    TriggL T0,v50,laserON,z0,toolEtna\WObj:=wobjEtna;
    TriggL T1,vl,laserOFF,z0,toolEtna\WObj:=wobjEtna;
    TriggL T2,v50,laserON,z0,toolEtna\WObj:=wobjEtna;
    TriggL T3,vl,laserOFF,z0,toolEtna\WObj:=wobjEtna;
    TriggL T4,v50,laserON,z0,toolEtna\WObj:=wobjEtna;
    TriggL T5,vl,laserOFF,z0,toolEtna\WObj:=wobjEtna;
    TriggL T6,v50,laserON,z0,toolEtna\WObj:=wobjEtna;
    TriggL T7,vl,laserOFF,z0,toolEtna\WObj:=wobjEtna;
    TriggL T8,v50,laserON,z0,toolEtna\WObj:=wobjEtna;
    TriggL T9,vl,laserOFF,z0,toolEtna\WObj:=wobjEtna;
    TriggL T10,v50,laserON,z0,toolEtna\WObj:=wobjEtna;
    TriggL T11,vl,laserOFF,z0,toolEtna\WObj:=wobjEtna;
    TriggL T12,v50,laserON,z0,toolEtna\WObj:=wobjEtna;
    TriggL T13,vl,laserOFF,z0,toolEtna\WObj:=wobjEtna;
    TriggL T14,v50,laserON,z0,toolEtna\WObj:=wobjEtna;
    TriggL T15,vl,laserOFF,z0,toolEtna\WObj:=wobjEtna;
    TriggL T16,v50,laserON,z0,toolEtna\WObj:=wobjEtna;
    TriggL T17,vl,laserOFF,z0,toolEtna\WObj:=wobjEtna;
    TriggL T18,v50,laserON,z0,toolEtna\WObj:=wobjEtna;
    TriggL T19,vl,laserOFF,z0,toolEtna\WObj:=wobjEtna;
    TriggL T20,v50,laserON,z0,toolEtna\WObj:=wobjEtna;
    TriggL T21,vl,laserOFF,z0,toolEtna\WObj:=wobjEtna;
    TriggL T22,v50,laserON,z0,toolEtna\WObj:=wobjEtna;
    TriggL T23,vl,laserOFF,z0,toolEtna\WObj:=wobjEtna;
    TriggL T24,v50,laserON,z0,toolEtna\WObj:=wobjEtna;
    TriggL T25,vl,laserOFF,z0,toolEtna\WObj:=wobjEtna;
    TriggL T26,v50,laserON,z0,toolEtna\WObj:=wobjEtna;
    TriggL T27,vl,laserOFF,z0,toolEtna\WObj:=wobjEtna;
    TriggL T28,v50,laserON,z0,toolEtna\WObj:=wobjEtna;
    TriggL T29,vl,laserOFF,z0,toolEtna\WObj:=wobjEtna;
    TriggL T30,v50,laserON,z0,toolEtna\WObj:=wobjEtna;
    TriggL T31,vl,laserOFF,z0,toolEtna\WObj:=wobjEtna;
    TriggL T32,v50,laserON,z0,toolEtna\WObj:=wobjEtna;
    TriggL T33,vl,laserOFF,z0,toolEtna\WObj:=wobjEtna;
    TriggL T34,v50,laserON,z0,toolEtna\WObj:=wobjEtna;
    TriggL T35,vl,laserOFF,z0,toolEtna\WObj:=wobjEtna;
    TriggL T36,v50,laserON,z0,toolEtna\WObj:=wobjEtna;
    TriggL T37,vl,laserOFF,z0,toolEtna\WObj:=wobjEtna;
    TriggL T38,v50,laserON,z0,toolEtna\WObj:=wobjEtna;
    TriggL T39,vl,laserOFF,z0,toolEtna\WObj:=wobjEtna;
    TriggL T40,v50,laserON,z0,toolEtna\WObj:=wobjEtna;
    TriggL T41,vl,laserOFF,z0,toolEtna\WObj:=wobjEtna;
    TriggL T42,v50,laserON,z0,toolEtna\WObj:=wobjEtna;
    TriggL T43,vl,laserOFF,z0,toolEtna\WObj:=wobjEtna;
    TriggL T44,v50,laserON,z0,toolEtna\WObj:=wobjEtna;
    TriggL T45,vl,laserOFF,z0,toolEtna\WObj:=wobjEtna;
    TriggL T46,v50,laserON,z0,toolEtna\WObj:=wobjEtna;
    TriggL T47,vl,laserOFF,z0,toolEtna\WObj:=wobjEtna;
    TriggL T48,v50,laserON,z0,toolEtna\WObj:=wobjEtna;
    TriggL T49,vl,laserOFF,z0,toolEtna\WObj:=wobjEtna;
    TriggL T50,v50,laserON,z0,toolEtna\WObj:=wobjEtna;
    TriggL T51,vl,laserOFF,z0,toolEtna\WObj:=wobjEtna;
    TriggL T52,v50,laserON,z0,toolEtna\WObj:=wobjEtna;
    TriggL T53,vl,laserOFF,z0,toolEtna\WObj:=wobjEtna;
    TriggL T54,v50,laserON,z0,toolEtna\WObj:=wobjEtna;
    TriggL T55,vl,laserOFF,z0,toolEtna\WObj:=wobjEtna;
    TriggL T56,v50,laserON,z0,toolEtna\WObj:=wobjEtna;
    TriggL T57,vl,laserOFF,z0,toolEtna\WObj:=wobjEtna;
    TriggL T58,v50,laserON,z0,toolEtna\WObj:=wobjEtna;
    TriggL T59,vl,laserOFF,z0,toolEtna\WObj:=wobjEtna;
    TriggL T60,v50,laserON,z0,toolEtna\WObj:=wobjEtna;
    TriggL T61,vl,laserOFF,z0,toolEtna\WObj:=wobjEtna;
    TriggL T62,v50,laserON,z0,toolEtna\WObj:=wobjEtna;
    TriggL T63,vl,laserOFF,z0,toolEtna\WObj:=wobjEtna;
    TriggL T64,v50,laserON,z0,toolEtna\WObj:=wobjEtna;
    TriggL T65,vl,laserOFF,z0,toolEtna\WObj:=wobjEtna;
    TriggL T66,v50,laserON,z0,toolEtna\WObj:=wobjEtna;
    TriggL T67,vl,laserOFF,z0,toolEtna\WObj:=wobjEtna;
    TriggL T68,v50,laserON,z0,toolEtna\WObj:=wobjEtna;
    TriggL T69,vl,laserOFF,z0,toolEtna\WObj:=wobjEtna;
    TriggL T70,v50,laserON,z0,toolEtna\WObj:=wobjEtna;
    TriggL T71,vl,laserOFF,z0,toolEtna\WObj:=wobjEtna;
    TriggL T72,v50,laserON,z0,toolEtna\WObj:=wobjEtna;
    TriggL T73,vl,laserOFF,z0,toolEtna\WObj:=wobjEtna;
    TriggL T74,v50,laserON,z0,toolEtna\WObj:=wobjEtna;
    TriggL T75,vl,laserOFF,z0,toolEtna\WObj:=wobjEtna;
    TriggL T76,v50,laserON,z0,toolEtna\WObj:=wobjEtna;
    TriggL T77,vl,laserOFF,z0,toolEtna\WObj:=wobjEtna;
    TriggL T78,v50,laserON,z0,toolEtna\WObj:=wobjEtna;
    TriggL T79,vl,laserOFF,z0,toolEtna\WObj:=wobjEtna;
    TriggL T80,v50,laserON,z0,toolEtna\WObj:=wobjEtna;
    TriggL T81,vl,laserOFF,z0,toolEtna\WObj:=wobjEtna;
    TriggL T82,v50,laserON,z0,toolEtna\WObj:=wobjEtna;
    TriggL T83,vl,laserOFF,z0,toolEtna\WObj:=wobjEtna;
    TriggL T84,v50,laserON,z0,toolEtna\WObj:=wobjEtna;
    TriggL T85,vl,laserOFF,z0,toolEtna\WObj:=wobjEtna;
    TriggL T86,v50,laserON,z0,toolEtna\WObj:=wobjEtna;
    TriggL T87,vl,laserOFF,z0,toolEtna\WObj:=wobjEtna;
    TriggL T88,v50,laserON,z0,toolEtna\WObj:=wobjEtna;
    TriggL T89,vl,laserOFF,z0,toolEtna\WObj:=wobjEtna;
    TriggL T90,v50,laserON,z0,toolEtna\WObj:=wobjEtna;
    TriggL T91,vl,laserOFF,z0,toolEtna\WObj:=wobjEtna;
    TriggL T92,v50,laserON,z0,toolEtna\WObj:=wobjEtna;
    TriggL T93,vl,laserOFF,z0,toolEtna\WObj:=wobjEtna;
    TriggL T94,v50,laserON,z0,toolEtna\WObj:=wobjEtna;
    TriggL T95,vl,laserOFF,z0,toolEtna\WObj:=wobjEtna;
    TriggL T96,v50,laserON,z0,toolEtna\WObj:=wobjEtna;
    TriggL T97,vl,laserOFF,z0,toolEtna\WObj:=wobjEtna;
    TriggL T98,v50,laserON,z0,toolEtna\WObj:=wobjEtna;
    TriggL T99,vl,laserOFF,z0,toolEtna\WObj:=wobjEtna;
    TriggL T100,v50,laserON,z0,toolEtna\WObj:=wobjEtna;
    TriggL T101,vl,laserOFF,z0,toolEtna\WObj:=wobjEtna;
    TriggL T102,v50,laserON,z0,toolEtna\WObj:=wobjEtna;
    TriggL T103,vl,laserOFF,z0,toolEtna\WObj:=wobjEtna;
    TriggL T104,v50,laserON,z0,toolEtna\WObj:=wobjEtna;
    TriggL T105,vl,laserOFF,z0,toolEtna\WObj:=wobjEtna;
    TriggL T106,v50,laserON,z0,toolEtna\WObj:=wobjEtna;
    TriggL T107,vl,laserOFF,z0,toolEtna\WObj:=wobjEtna;
    TriggL T108,v50,laserON,z0,toolEtna\WObj:=wobjEtna;
    TriggL T109,vl,laserOFF,z0,toolEtna\WObj:=wobjEtna;
    TriggL T110,v50,laserON,z0,toolEtna\WObj:=wobjEtna;
    TriggL T111,vl,laserOFF,z0,toolEtna\WObj:=wobjEtna;
    TriggL T112,v50,laserON,z0,toolEtna\WObj:=wobjEtna;
    TriggL T113,vl,laserOFF,z0,toolEtna\WObj:=wobjEtna;
    TriggL T114,v50,laserON,z0,toolEtna\WObj:=wobjEtna;
    TriggL T115,vl,laserOFF,z0,toolEtna\WObj:=wobjEtna;
    TriggL T116,v50,laserON,z0,toolEtna\WObj:=wobjEtna;
    TriggL T117,vl,laserOFF,z0,toolEtna\WObj:=wobjEtna;
    TriggL T118,v50,laserON,z0,toolEtna\WObj:=wobjEtna;
    TriggL T119,vl,laserOFF,z0,toolEtna\WObj:=wobjEtna;
    TriggL T120,v50,laserON,z0,toolEtna\WObj:=wobjEtna;
    TriggL T121,vl,laserOFF,z0,toolEtna\WObj:=wobjEtna;
    TriggL T122,v50,laserON,z0,toolEtna\WObj:=wobjEtna;
    TriggL T123,vl,laserOFF,z0,toolEtna\WObj:=wobjEtna;
    TriggL T124,v50,laserON,z0,toolEtna\WObj:=wobjEtna;
    TriggL T125,vl,laserOFF,z0,toolEtna\WObj:=wobjEtna;
    TriggL T126,v50,laserON,z0,toolEtna\WObj:=wobjEtna;
    TriggL T127,vl,laserOFF,z0,toolEtna\WObj:=wobjEtna;
    TriggL T128,v50,laserON,z0,toolEtna\WObj:=wobjEtna;
    TriggL T129,vl,laserOFF,z0,toolEtna\WObj:=wobjEtna;
    TriggL T130,v50,laserON,z0,toolEtna\WObj:=wobjEtna;
    TriggL T131,vl,laserOFF,z0,toolEtna\WObj:=wobjEtna;
    TriggL T132,v50,laserON,z0,toolEtna\WObj:=wobjEtna;
    TriggL T133,vl,laserOFF,z0,toolEtna\WObj:=wobjEtna;
    TriggL T134,v50,laserON,z0,toolEtna\WObj:=wobjEtna;
    TriggL T135,vl,laserOFF,z0,toolEtna\WObj:=wobjEtna;
    TriggL T136,v50,laserON,z0,toolEtna\WObj:=wobjEtna;
    TriggL T137,vl,laserOFF,z0,toolEtna\WObj:=wobjEtna;
    TriggL T138,v50,laserON,z0,toolEtna\WObj:=wobjEtna;
    TriggL T139,vl,laserOFF,z0,toolEtna\WObj:=wobjEtna;
    TriggL T140,v50,laserON,z0,toolEtna\WObj:=wobjEtna;
    TriggL T141,vl,laserOFF,z0,toolEtna\WObj:=wobjEtna;
    TriggL T142,v50,laserON,z0,toolEtna\WObj:=wobjEtna;
    TriggL T143,vl,laserOFF,z0,toolEtna\WObj:=wobjEtna;
    TriggL T144,v50,laserON,z0,toolEtna\WObj:=wobjEtna;
    TriggL T145,vl,laserOFF,z0,toolEtna\WObj:=wobjEtna;
    TriggL T146,v50,laserON,z0,toolEtna\WObj:=wobjEtna;
    TriggL T147,vl,laserOFF,z0,toolEtna\WObj:=wobjEtna;
    TriggL T148,v50,laserON,z0,toolEtna\WObj:=wobjEtna;
    TriggL T149,vl,laserOFF,z0,toolEtna\WObj:=wobjEtna;
    TriggL T150,v50,laserON,z0,toolEtna\WObj:=wobjEtna;
    TriggL T151,vl,laserOFF,z0,toolEtna\WObj:=wobjEtna;
    TriggL T152,v50,laserON,z0,toolEtna\WObj:=wobjEtna;
    TriggL T153,vl,laserOFF,z0,toolEtna\WObj:=wobjEtna;
    TriggL T154,v50,laserON,z0,toolEtna\WObj:=wobjEtna;
    TriggL T155,vl,laserOFF,z0,toolEtna\WObj:=wobjEtna;
    TriggL T156,v50,laserON,z0,toolEtna\WObj:=wobjEtna;
    TriggL T157,vl,laserOFF,z0,toolEtna\WObj:=wobjEtna;
    TriggL T158,v50,laserON,z0,toolEtna\WObj:=wobjEtna;
    TriggL T159,vl,laserOFF,z0,toolEtna\WObj:=wobjEtna;
    TriggL T160,v50,laserON,z0,toolEtna\WObj:=wobjEtna;
    TriggL T161,vl,laserOFF,z0,toolEtna\WObj:=wobjEtna;
    TriggL T162,v50,laserON,z0,toolEtna\WObj:=wobjEtna;
    TriggL T163,vl,laserOFF,z0,toolEtna\WObj:=wobjEtna;
    TriggL T164,v50,laserON,z0,toolEtna\WObj:=wobjEtna;
    TriggL T165,vl,laserOFF,z0,toolEtna\WObj:=wobjEtna;
    TriggL T166,v50,laserON,z0,toolEtna\WObj:=wobjEtna;
    TriggL T167,vl,laserOFF,z0,toolEtna\WObj:=wobjEtna;
    TriggL T168,v50,laserON,z0,toolEtna\WObj:=wobjEtna;
    TriggL T169,vl,laserOFF,z0,toolEtna\WObj:=wobjEtna;
    TriggL T170,v50,laserON,z0,toolEtna\WObj:=wobjEtna;
    TriggL T171,vl,laserOFF,z0,toolEtna\WObj:=wobjEtna;
    TriggL T172,v50,laserON,z0,toolEtna\WObj:=wobjEtna;
    TriggL T173,vl,laserOFF,z0,toolEtna\WObj:=wobjEtna;
    TriggL T174,v50,laserON,z0,toolEtna\WObj:=wobjEtna;
    TriggL T175,vl,laserOFF,z0,toolEtna\WObj:=wobjEtna;
    TriggL T176,v50,laserON,z0,toolEtna\WObj:=wobjEtna;
    TriggL T177,vl,laserOFF,z0,toolEtna\WObj:=wobjEtna;
    TriggL T178,v50,laserON,z0,toolEtna\WObj:=wobjEtna;
    TriggL T179,vl,laserOFF,z0,toolEtna\WObj:=wobjEtna;
    TriggL T180,v50,laserON,z0,toolEtna\WObj:=wobjEtna;
    TriggL T181,vl,laserOFF,z0,toolEtna\WObj:=wobjEtna;
    TriggL T182,v50,laserON,z0,toolEtna\WObj:=wobjEtna;
    TriggL T183,vl,laserOFF,z0,toolEtna\WObj:=wobjEtna;
    TriggL T184,v50,laserON,z0,toolEtna\WObj:=wobjEtna;
    TriggL T185,vl,laserOFF,z0,toolEtna\WObj:=wobjEtna;
    TriggL T186,v50,laserON,z0,toolEtna\WObj:=wobjEtna;
    TriggL T187,vl,laserOFF,z0,toolEtna\WObj:=wobjEtna;
    TriggL T188,v50,laserON,z0,toolEtna\WObj:=wobjEtna;
    TriggL T189,vl,laserOFF,z0,toolEtna\WObj:=wobjEtna;
    TriggL T190,v50,laserON,z0,toolEtna\WObj:=wobjEtna;
    TriggL T191,vl,laserOFF,z0,toolEtna\WObj:=wobjEtna;
    TriggL T192,v50,laserON,z0,toolEtna\WObj:=wobjEtna;
    TriggL T193,vl,laserOFF,z0,toolEtna\WObj:=wobjEtna;
    TriggL T194,v50,laserON,z0,toolEtna\WObj:=wobjEtna;
    TriggL T195,vl,laserOFF,z0,toolEtna\WObj:=wobjEtna;
    TriggL T196,v50,laserON,z0,toolEtna\WObj:=wobjEtna;
    TriggL T197,vl,laserOFF,z0,toolEtna\WObj:=wobjEtna;
    TriggL T198,v50,laserON,z0,toolEtna\WObj:=wobjEtna;
    TriggL T199,vl,laserOFF,z0,toolEtna\WObj:=wobjEtna;
    TriggL T200,v50,laserON,z0,toolEtna\WObj:=wobjEtna;
    TriggL T201,vl,laserOFF,z0,toolEtna\WObj:=wobjEtna;
    TriggL T202,v50,laserON,z0,toolEtna\WObj:=wobjEtna;
    TriggL T203,vl,laserOFF,z0,toolEtna\WObj:=wobjEtna;
    TriggL T204,v50,laserON,z0,toolEtna\WObj:=wobjEtna;
    TriggL T205,vl,laserOFF,z0,toolEtna\WObj:=wobjEtna;
    TriggL T206,v50,laserON,z0,toolEtna\WObj:=wobjEtna;
    TriggL T207,vl,laserOFF,z0,toolEtna\WObj:=wobjEtna;
    TriggL T208,v50,laserON,z0,toolEtna\WObj:=wobjEtna;
    TriggL T209,vl,laserOFF,z0,toolEtna\WObj:=wobjEtna;
    TriggL T210,v50,laserON,z0,toolEtna\WObj:=wobjEtna;
    TriggL T211,vl,laserOFF,z0,toolEtna\WObj:=wobjEtna;
    TriggL T212,v50,laserON,z0,toolEtna\WObj:=wobjEtna;
    TriggL T213,vl,laserOFF,z0,toolEtna\WObj:=wobjEtna;
    TriggL T214,v50,laserON,z0,toolEtna\WObj:=wobjEtna;
    TriggL T215,vl,laserOFF,z0,toolEtna\WObj:=wobjEtna;
    TriggL T216,v50,laserON,z0,toolEtna\WObj:=wobjEtna;
    TriggL T217,vl,laserOFF,z0,toolEtna\WObj:=wobjEtna;
    TriggL T218,v50,laserON,z0,toolEtna\WObj:=wobjEtna;
    TriggL T219,vl,laserOFF,z0,toolEtna\WObj:=wobjEtna;
    TriggL T220,v50,laserON,z0,toolEtna\WObj:=wobjEtna;
    TriggL T221,vl,laserOFF,z0,toolEtna\WObj:=wobjEtna;
    TriggL T222,v50,laserON,z0,toolEtna\WObj:=wobjEtna;
    TriggL T223,vl,laserOFF,z0,toolEtna\WObj:=wobjEtna;
    TriggL T224,v50,laserON,z0,toolEtna\WObj:=wobjEtna;
    TriggL T225,vl,laserOFF,z0,toolEtna\WObj:=wobjEtna;
    TriggL T226,v50,laserON,z0,toolEtna\WObj:=wobjEtna;
    TriggL T227,vl,laserOFF,z0,toolEtna\WObj:=wobjEtna;
    TriggL T228,v50,laserON,z0,toolEtna\WObj:=wobjEtna;
    TriggL T229,vl,laserOFF,z0,toolEtna\WObj:=wobjEtna;
    TriggL T230,v50,laserON,z0,toolEtna\WObj:=wobjEtna;
    TriggL T231,vl,laserOFF,z0,toolEtna\WObj:=wobjEtna;
    TriggL T232,v50,laserON,z0,toolEtna\WObj:=wobjEtna;
    TriggL T233,vl,laserOFF,z0,toolEtna\WObj:=wobjEtna;
    TriggL T234,v50,laserON,z0,toolEtna\WObj:=wobjEtna;
    TriggL T235,vl,laserOFF,z0,toolEtna\WObj:=wobjEtna;
    TriggL T236,v50,laserON,z0,toolEtna\WObj:=wobjEtna;
    TriggL T237,vl,laserOFF,z0,toolEtna\WObj:=wobjEtna;
    TriggL T238,v50,laserON,z0,toolEtna\WObj:=wobjEtna;
    TriggL T239,vl,laserOFF,z0,toolEtna\WObj:=wobjEtna;
    TriggL T240,v50,laserON,z0,toolEtna\WObj:=wobjEtna;
    TriggL T241,vl,laserOFF,z0,toolEtna\WObj:=wobjEtna;
    TriggL T242,v50,laserON,z0,toolEtna\WObj:=wobjEtna;
    TriggL T243,vl,laserOFF,z0,toolEtna\WObj:=wobjEtna;
    TriggL T244,v50,laserON,z0,toolEtna\WObj:=wobjEtna;
    TriggL T245,vl,laserOFF,z0,toolEtna\WObj:=wobjEtna;
    TriggL T246,v50,laserON,z0,toolEtna\WObj:=wobjEtna;
    TriggL T247,vl,laserOFF,z0,toolEtna\WObj:=wobjEtna;
    TriggL T248,v50,laserON,z0,toolEtna\WObj:=wobjEtna;
    TriggL T249,vl,laserOFF,z0,toolEtna\WObj:=wobjEtna;
    TriggL T250,v50,laserON,z0,toolEtna\WObj:=wobjEtna;
    TriggL T251,vl,laserOFF,z0,toolEtna\WObj:=wobjEtna;
    TriggL T252,v50,laserON,z0,toolEtna\WObj:=wobjEtna;
    TriggL T253,vl,laserOFF,z0,toolEtna\WObj:=wobjEtna;
    TriggL T254,v50,laserON,z0,toolEtna\WObj:=wobjEtna;
    TriggL T255,vl,laserOFF,z0,toolEtna\WObj:=wobjEtna;
    TriggL T256,v50,laserON,z0,toolEtna\WObj:=wobjEtna;
    TriggL T257,vl,laserOFF,z0,toolEtna\WObj:=wobjEtna;
    TriggL T258,v50,laserON,z0,toolEtna\WObj:=wobjEtna;
    TriggL T259,vl,laserOFF,z0,toolEtna\WObj:=wobjEtna;
    TriggL T260,v50,laserON,z0,toolEtna\WObj:=wobjEtna;
    TriggL T261,vl,laserOFF,z0,toolEtna\WObj:=wobjEtna;
    TriggL T262,v50,laserON,z0,toolEtna\WObj:=wobjEtna;
    TriggL T263,vl,laserOFF,z0,toolEtna\WObj:=wobjEtna;
    TriggL T264,v50,laserON,z0,toolEtna\WObj:=wobjEtna;
    TriggL T265,vl,laserOFF,z0,toolEtna\WObj:=wobjEtna;
    TriggL T266,v50,laserON,z0,toolEtna\WObj:=wobjEtna;
    TriggL T267,vl,laserOFF,z0,toolEtna\WObj:=wobjEtna;
    TriggL T268,v50,laserON,z0,toolEtna\WObj:=wobjEtna;
    TriggL T269,vl,laserOFF,z0,toolEtna\WObj:=wobjEtna;
    TriggL T270,v50,laserON,z0,toolEtna\WObj:=wobjEtna;
    TriggL T271,vl,laserOFF,z0,toolEtna\WObj:=wobjEtna;
    TriggL T272,v50,laserON,z0,toolEtna\WObj:=wobjEtna;
    TriggL T273,vl,laserOFF,z0,toolEtna\WObj:=wobjEtna;
    TriggL T274,v50,laserON,z0,toolEtna\WObj:=wobjEtna;
    TriggL T275,vl,laserOFF,z0,toolEtna\WObj:=wobjEtna;
    TriggL T276,v50,laserON,z0,toolEtna\WObj:=wobjEtna;
    TriggL T277,vl,laserOFF,z0,toolEtna\WObj:=wobjEtna;
    TriggL T278,v50,laserON,z0,toolEtna\WObj:=wobjEtna;
    TriggL T279,vl,laserOFF,z0,toolEtna\WObj:=wobjEtna;
    TriggL T280,v50,laserON,z0,toolEtna\WObj:=wobjEtna;
    TriggL T281,vl,laserOFF,z0,toolEtna\WObj:=wobjEtna;
    TriggL T282,v50,laserON,z0,toolEtna\WObj:=wobjEtna;
    TriggL T283,vl,laserOFF,z0,toolEtna\WObj:=wobjEtna;
    TriggL T284,v50,laserON,z0,toolEtna\WObj:=wobjEtna;
    TriggL T285,vl,laserOFF,z0,toolEtna\WObj:=wobjEtna;
    TriggL T286,v50,laserON,z0,toolEtna\WObj:=wobjEtna;
    TriggL T287,vl,laserOFF,z0,toolEtna\WObj:=wobjEtna;
    TriggL T288,v50,laserON,z0,toolEtna\WObj:=wobjEtna;
    TriggL T289,vl,laserOFF,z0,toolEtna\WObj:=wobjEtna;
    TriggL T290,v50,laserON,z0,toolEtna\WObj:=wobjEtna;
    TriggL T291,vl,laserOFF,z0,toolEtna\WObj:=wobjEtna;
    TriggL T292,v50,laserON,z0,toolEtna\WObj:=wobjEtna;
    TriggL T293,vl,laserOFF,z0,toolEtna\WObj:=wobjEtna;
    TriggL T294,v50,laserON,z0,toolEtna\WObj:=wobjEtna;
    TriggL T295,vl,laserOFF,z0,toolEtna\WObj:=wobjEtna;
    TriggL T296,v50,laserON,z0,toolEtna\WObj:=wobjEtna;
    TriggL T297,vl,laserOFF,z0,toolEtna\WObj:=wobjEtna;
    TriggL T298,v50,laserON,z0,toolEtna\WObj:=wobjEtna;
    TriggL T299,vl,laserOFF,z0,toolEtna\WObj:=wobjEtna;
    TriggL T300,v50,laserON,z0,toolEtna\WObj:=wobjEtna;
    TriggL T301,vl,laserOFF,z0,toolEtna\WObj:=wobjEtna;
    TriggL T302,v50,laserON,z0,toolEtna\WObj:=wobjEtna;
    TriggL T303,vl,laserOFF,z0,toolEtna\WObj:=wobjEtna;
    TriggL T304,v50,laserON,z0,toolEtna\WObj:=wobjEtna;
    TriggL T305,vl,laserOFF,z0,toolEtna\WObj:=wobjEtna;
    TriggL T306,v50,laserON,z0,toolEtna\WObj:=wobjEtna;
    TriggL T307,vl,laserOFF,z0,toolEtna\WObj:=wobjEtna;
    TriggL T308,v50,laserON,z0,toolEtna\WObj:=wobjEtna;
    TriggL T309,vl,laserOFF,z0,toolEtna\WObj:=wobjEtna;
    TriggL T310,v50,laserON,z0,toolEtna\WObj:=wobjEtna;
    TriggL T311,vl,laserOFF,z0,toolEtna\WObj:=wobjEtna;
    TriggL T312,v50,laserON,z0,toolEtna\WObj:=wobjEtna;
    TriggL T313,vl,laserOFF,z0,toolEtna\WObj:=wobjEtna;
    TriggL T314,v50,laserON,z0,toolEtna\WObj:=wobjEtna;
    TriggL T315,vl,laserOFF,z0,toolEtna\WObj:=wobjEtna;
    TriggL T316,v50,laserON,z0,toolEtna\WObj:=wobjEtna;
    TriggL T317,vl,laserOFF,z0,toolEtna\WObj:=wobjEtna;
    TriggL T318,v50,laserON,z0,toolEtna\WObj:=wobjEtna;
    TriggL T319,vl,laserOFF,z0,toolEtna\WObj:=wobjEtna;
    TriggL T320,v50,laserON,z0,toolEtna\WObj:=wobjEtna;
    TriggL T321,vl,laserOFF,z0,toolEtna\WObj:=wobjEtna;
    TriggL T322,v50,laserON,z0,toolEtna\WObj:=wobjEtna;
    TriggL T323,vl,laserOFF,z0,toolEtna\WObj:=wobjEtna;
    TriggL T324,v50,laserON,z0,toolEtna\WObj:=wobjEtna;
    TriggL T325,vl,laserOFF,z0,toolEtna\WObj:=wobjEtna;
    TriggL T326,v50,laserON,z0,toolEtna\WObj:=wobjEtna;
    TriggL T327,vl,laserOFF,z0,toolEtna\WObj:=wobjEtna;
    TriggL T328,v50,laserON,z0,toolEtna\WObj:=wobjEtna;
    TriggL T329,vl,laserOFF,z0,toolEtna\WObj:=wobjEtna;
    TriggL T330,v50,laserON,z0,toolEtna\WObj:=wobjEtna;
    TriggL T331,vl,laserOFF,z0,toolEtna\WObj:=wobjEtna;
    TriggL T332,v50,laserON,z0,toolEtna\WObj:=wobjEtna;
    TriggL T333,vl,laserOFF,z0,toolEtna\WObj:=wobjEtna;
    TriggL T334,v50,laserON,z0,toolEtna\WObj:=wobjEtna;
    TriggL T335,vl,laserOFF,z0,toolEtna\WObj:=wobjEtna;
    TriggL T336,v50,laserON,z0,toolEtna\WObj:=wobjEtna;
    TriggL T337,vl,laserOFF,z0,toolEtna\WObj:=wobjEtna;
    TriggL T338,v50,laserON,z0,toolEtna\WObj:=wobjEtna;
    TriggL T339,vl,laserOFF,z0,toolEtna\WObj:=wobjEtna;
    TriggL T340,v50,laserON,z0,toolEtna\WObj:=wobjEtna;
    TriggL T341,vl,laserOFF,z0,toolEtna\WObj:=wobjEtna;
    TriggL T342,v50,laserON,z0,toolEtna\WObj:=wobjEtna;
    TriggL T343,vl,laserOFF,z0,toolEtna\WObj:=wobjEtna;
    TriggL T344,v50,laserON,z0,toolEtna\WObj:=wobjEtna;
    TriggL T345,vl,laserOFF,z0,toolEtna\WObj:=wobjEtna;
    TriggL T346,v50,laserON,z0,toolEtna\WObj:=wobjEtna;
    TriggL T347,vl,laserOFF,z0,toolEtna\WObj:=wobjEtna;
    TriggL T348,v50,laserON,z0,toolEtna\WObj:=wobjEtna;
    TriggL T349,vl,laserOFF,z0,toolEtna\WObj:=wobjEtna;
    TriggL T350,v50,laserON,z0,toolEtna\WObj:=wobjEtna;
    TriggL T351,vl,laserOFF,z0,toolEtna\WObj:=wobjEtna;
    TriggL T352,v50,laserON,z0,toolEtna\WObj:=wobjEtna;
    TriggL T353,vl,laserOFF,z0,toolEtna\WObj:=wobjEtna;
    TriggL T354,v50,laserON,z0,toolEtna\WObj:=wobjEtna;
    TriggL T355,vl,laserOFF,z0,toolEtna\WObj:=wobjEtna;
    TriggL T356,v50,laserON,z0,toolEtna\WObj:=wobjEtna;
    TriggL T357,vl,laserOFF,z0,toolEtna\WObj:=wobjEtna;
    TriggL T358,v50,laserON,z0,toolEtna\WObj:=wobjEtna;
    TriggL T359,vl,laserOFF,z0,toolEtna\WObj:=wobjEtna;
    TriggL T360,v50,laserON,z0,toolEtna\WObj:=wobjEtna;
    TriggL T361,vl,laserOFF,z0,toolEtna\WObj:=wobjEtna;
    TriggL T362,v50,laserON,z0,toolEtna\WObj:=wobjEtna;
    TriggL T363,vl,laserOFF,z0,toolEtna\WObj:=wobjEtna;
    TriggL T364,v50,laserON,z0,toolEtna\WObj:=wobjEtna;
    TriggL T365,vl,laserOFF,z0,toolEtna\WObj:=wobjEtna;
    TriggL T366,v50,laserON,z0,toolEtna\WObj:=wobjEtna;
    TriggL T367,vl,laserOFF,z0,toolEtna\WObj:=wobjEtna;
    TriggL T368,v50,laserON,z0,toolEtna\WObj:=wobjEtna;
    TriggL T369,vl,laserOFF,z0,toolEtna\WObj:=wobjEtna;
    TriggL T370,v50,laserON,z0,toolEtna\WObj:=wobjEtna;
    TriggL T371,vl,laserOFF,z0,toolEtna\WObj:=wobjEtna;
    TriggL T372,v50,laserON,z0,toolEtna\WObj:=wobjEtna;
    TriggL T373,vl,laserOFF,z0,toolEtna\WObj:=wobjEtna;
    TriggL T374,v50,laserON,z0,toolEtna\WObj:=wobjEtna;
    TriggL T375,vl,laserOFF,z0,toolEtna\WObj:=wobjEtna;
    TriggL T376,v50,laserON,z0,toolEtna\WObj:=wobjEtna;
    TriggL T377,vl,laserOFF,z0,toolEtna\WObj:=wobjEtna;
    TriggL T378,v50,laserON,z0,toolEtna\WObj:=wobjEtna;
    TriggL T379,vl,laserOFF,z0,toolEtna\WObj:=wobjEtna;
    TriggL T380,v50,laserON,z0,toolEtna\WObj:=wobjEtna;
    TriggL T381,vl,laserOFF,z0,toolEtna\WObj:=wobjEtna;
    TriggL T382,v50,laserON,z0,toolEtna\WObj:=wobjEtna;
    TriggL T383,vl,laserOFF,z0,toolEtna\WObj:=wobjEtna;
    TriggL T384,v50,laserON,z0,toolEtna\WObj:=wobjEtna;
    TriggL T385,vl,laserOFF,z0,toolEtna\WObj:=wobjEtna;
    TriggL T386,v50,laserON,z0,toolEtna\WObj:=wobjEtna;
    TriggL T387,vl,laserOFF,z0,toolEtna\WObj:=wobjEtna;
    TriggL T388,v50,laserON,z0,toolEtna\WObj:=wobjEtna;
    TriggL T389,vl,laserOFF,z0,toolEtna\WObj:=wobjEtna;
    TriggL T390,v50,laserON,z0,toolEtna\WObj:=wobjEtna;
    TriggL T391,vl,laserOFF,z0,toolEtna\WObj:=wobjEtna;
    TriggL T392,v50,laserON,z0,toolEtna\WObj:=wobjEtna;
    TriggL T393,vl,laserOFF,z0,toolEtna\WObj:=wobjEtna;
    TriggL T394,v50,laserON,z0,toolEtna\WObj:=wobjEtna;
    TriggL T395,vl,laserOFF,z0,toolEtna\WObj:=wobjEtna;
    TriggL T396,v50,laserON,z0,toolEtna\WObj:=wobjEtna;
    TriggL T397,vl,laserOFF,z0,toolEtna\WObj:=wobjEtna;
    TriggL T398,v50,laserON,z0,toolEtna\WObj:=wobjEtna;
    TriggL T399,vl,laserOFF,z0,toolEtna\WObj:=wobjEtna;
    TriggL T400,v50,laserON,z0,toolEtna\WObj:=wobjEtna;
    TriggL T401,vl,laserOFF,z0,toolEtna\WObj:=wobjEtna;
    TriggL T402,v50,laserON,z0,toolEtna\WObj:=wobjEtna;
    TriggL T403,vl,laserOFF,z0,toolEtna\WObj:=wobjEtna;
    TriggL T404,v50,laserON,z0,toolEtna\WObj:=wobjEtna;
    TriggL T405,vl,laserOFF,z0,toolEtna\WObj:=wobjEtna;
    TriggL T406,v50,laserON,z0,toolEtna\WObj:=wobjEtna;
    TriggL T407,vl,laserOFF,z0,toolEtna\WObj:=wobjEtna;
    TriggL T408,v50,laserON,z0,toolEtna\WObj:=wobjEtna;
    TriggL T409,vl,laserOFF,z0,toolEtna\WObj:=wobjEtna;
    TriggL T410,v50,laserON,z0,toolEtna\WObj:=wobjEtna;
    TriggL T411,vl,laserOFF,z0,toolEtna\WObj:=wobjEtna;
    TriggL T412,v50,laserON,z0,toolEtna\WObj:=wobjEtna;
    TriggL T413,vl,laserOFF,z0,toolEtna\WObj:=wobjEtna;
    TriggL T414,v50,laserON,z0,toolEtna\WObj:=wobjEtna;
    TriggL T415,vl,laserOFF,z0,toolEtna\WObj:=wobjEtna;
    TriggL T416,v50,laserON,z0,toolEtna\WObj:=wobjEtna;
    TriggL T417,vl,laserOFF,z0,toolEtna\WObj:=wobjEtna;
    TriggL T418,v50,laserON,z0,toolEtna\WObj:=wobjEtna;
    TriggL T419,vl,laserOFF,z0,toolEtna\WObj:=wobjEtna;
    TriggL T420,v50,laserON,z0,toolEtna\WObj:=wobjEtna;
    TriggL T421,vl,laserOFF,z0,toolEtna\WObj:=wobjEtna;
    TriggL T422,v50,laserON,z0,toolEtna\WObj:=wobjEtna;
    TriggL T423,vl,laserOFF,z0,toolEtna\WObj:=wobjEtna;
    TriggL T424,v50,laserON,z0,toolEtna\WObj:=wobjEtna;
    TriggL T425,vl,laserOFF,z0,toolEtna\WObj:=wobjEtna;
    TriggL T426,v50,laserON,z0,toolEtna\WObj:=wobjEtna;
    TriggL T427,vl,laserOFF,z0,toolEtna\WObj:=wobjEtna;
    TriggL T428,v50,laserON,z0,toolEtna\WObj:=wobjEtna;
    TriggL T429,vl,laserOFF,z0,toolEtna\WObj:=wobjEtna;
    TriggL T430,v50,laserON,z0,toolEtna\WObj:=wobjEtna;
    TriggL T431,vl,laserOFF,z0,toolEtna\WObj:=wobjEtna;
    TriggL T432,v50,laserON,z0,toolEtna\WObj:=wobjEtna;
    TriggL T433,vl,laserOFF,z0,toolEtna\WObj:=wobjEtna;
    TriggL T434,v50,laserON,z0,toolEtna\WObj:=wobjEtna;
    TriggL T435,vl,laserOFF,z0,toolEtna\WObj:=wobjEtna;
    TriggL T436,v50,laserON,z0,toolEtna\WObj:=wobjEtna;
    TriggL T437,vl,laserOFF,z0,toolEtna\WObj:=wobjEtna;
    TriggL T438,v50,laserON,z0,toolEtna\WObj:=wobjEtna;
    TriggL T439,vl,laserOFF,z0,toolEtna\WObj:=wobjEtna;
    TriggL T440,v50,laserON,z0,toolEtna\WObj:=wobjEtna;
    TriggL T441,vl,laserOFF,z0,toolEtna\WObj:=wobjEtna;
    TriggL T442,v50,laserON,z0,toolEtna\WObj:=wobjEtna;
    TriggL T443,vl,laserOFF,z0,toolEtna\WObj:=wobjEtna;
    TriggL T444,v50,laserON,z0,toolEtna\WObj:=wobjEtna;
    TriggL T445,vl,laserOFF,z0,toolEtna\WObj:=wobjEtna;
    TriggL T446,v50,laserON,z0,toolEtna\WObj:=wobjEtna;
    TriggL T447,vl,laserOFF,z0,toolEtna\WObj:=wobjEtna;
    TriggL T448,v50,laserON,z0,toolEtna\WObj:=wobjEtna;
    TriggL T449,vl,laserOFF,z0,toolEtna\WObj:=wobjEtna;
    TriggL T450,v50,laserON,z0,toolEtna\WObj:=wobjEtna;
    TriggL T451,vl,laserOFF,z0,toolEtna\WObj:=wobjEtna;
    TriggL T452,v50,laserON,z0,toolEtna\WObj:=wobjEtna;
    TriggL T453,vl,laserOFF,z0,toolEtna\WObj:=wobjEtna;
    TriggL T454,v50,laserON,z0,toolEtna\WObj:=wobjEtna;
    TriggL T455,vl,laserOFF,z0,toolEtna\WObj:=wobjEtna;
    TriggL T456,v50,laserON,z0,toolEtna\WObj:=wobjEtna;
    TriggL T457,vl,laserOFF,z0,toolEtna\WObj:=wobjEtna;
    TriggL T458,v50,laserON,z0,toolEtna\WObj:=wobjEtna;
    TriggL T459,vl,laserOFF,z0,toolEtna\WObj:=wobjEtna;
    TriggL T460,v50,laserON,z0,toolEtna\WObj:=wobjEtna;
    TriggL T461,vl,laserOFF,z0,toolEtna\WObj:=wobjEtna;
    TriggL T462,v50,laserON,z0,toolEtna\WObj:=wobjEtna;
    TriggL T463,vl,laserOFF,z0,toolEtna\WObj:=wobjEtna;
    TriggL T464,v50,laserON,z0,toolEtna\WObj:=wobjEtna;
    TriggL T465,vl,laserOFF,z0,toolEtna\WObj:=wobjEtna;
    TriggL T466,v50,laserON,z0,toolEtna\WObj:=wobjEtna;
    TriggL T467,vl,laserOFF,z0,toolEtna\WObj:=wobjEtna;
    TriggL T468,v50,laserON,z0,toolEtna\WObj:=wobjEtna;
    TriggL T469,vl,laserOFF,z0,toolEtna\WObj:=wobjEtna;
    TriggL T470,v50,laserON,z0,toolEtna\WObj:=wobjEtna;
    TriggL T471,vl,laserOFF,z0,toolEtna\WObj:=wobjEtna;
    TriggL T472,v50,laserON,z0,toolEtna\WObj:=wobjEtna;
    TriggL T473,vl,laserOFF,z0,toolEtna\WObj:=wobjEtna;
    TriggL T474,v50,laserON,z0,toolEtna\WObj:=wobjEtna;
    TriggL T475,vl,laserOFF,z0,toolEtna\WObj:=wobjEtna;
    TriggL T476,v50,laserON,z0,toolEtna\WObj:=wobjEtna;
    TriggL T477,vl,laserOFF,z0,toolEtna\WObj:=wobjEtna;
    TriggL T478,v50,laserON,z0,toolEtna\WObj:=wobjEtna;
    TriggL T479,vl,laserOFF,z0,toolEtna\WObj:=wobjEtna;
    TriggL T480,v50,laserON,z0,toolEtna\WObj:=wobjEtna;
    TriggL T481,vl,laserOFF,z0,toolEtna\WObj:=wobjEtna;
    TriggL T482,v50,laserON,z0,toolEtna\WObj:=wobjEtna;
    TriggL T483,vl,laserOFF,z0,toolEtna\WObj:=wobjEtna;
    TriggL T484,v50,laserON,z0,toolEtna\WObj:=wobjEtna;
    TriggL T485,vl,laserOFF,z0,toolEtna\WObj:=wobjEtna;
    TriggL T486,v50,laserON,z0,toolEtna\WObj:=wobjEtna;
    TriggL T487,vl,laserOFF,z0,toolEtna\WObj:=wobjEtna;
    TriggL T488,v50,laserON,z0,toolEtna\WObj:=wobjEtna;
    TriggL T489,vl,laserOFF,z0,toolEtna\WObj:=wobjEtna;
    TriggL T490,v50,laserON,z0,toolEtna\WObj:=wobjEtna;
    TriggL T491,vl,laserOFF,z0,toolEtna\WObj:=wobjEtna;
    TriggL T492,v50,laserON,z0,toolEtna\WObj:=wobjEtna;
    TriggL T493,vl,laserOFF,z0,toolEtna\WObj:=wobjEtna;
    TriggL T494,v50,laserON,z0,toolEtna\WObj:=wobjEtna;
    TriggL T495,vl,laserOFF,z0,toolEtna\WObj:=wobjEtna;
    TriggL T496,v50,laserON,z0,toolEtna\WObj:=wobjEtna;
    TriggL T497,vl,laserOFF,z0,toolEtna\WObj:=wobjEtna;
    TriggL T498,v50,laserON,z0,toolEtna\WObj:=wobjEtna;
    TriggL T499,vl,laserOFF,z0,toolEtna\WObj:=wobjEtna;
    TriggL T500,v50,laserON,z0,toolEtna\WObj:=wobjEtna;
    TriggL T501,vl,laserOFF,z0,toolEtna\WObj:=wobjEtna;
    TriggL T502,v50,laserON,z0,toolEtna\WObj:=wobjEtna;
    TriggL T503,vl,laserOFF,z0,toolEtna\WObj:=wobjEtna;
    TriggL T504,v50,laserON,z0,toolEtna\WObj:=wobjEtna;
    TriggL T505,vl,laserOFF,z0,toolEtna\WObj:=wobjEtna;
    TriggL T506,v50,laserON,z0,toolEtna\WObj:=wobjEtna;
    TriggL T507,vl,laserOFF,z0,toolEtna\WObj:=wobjEtna;
    TriggL T508,v50,laserON,z0,toolEtna\WObj:=wobjEtna;
    TriggL T509,vl,laserOFF,z0,toolEtna\WObj:=wobjEtna;
    TriggL T510,v50,laserON,z0,toolEtna\WObj:=wobjEtna;
    TriggL T511,vl,laserOFF,z0,toolEtna\WObj:=wobjEtna;
    TriggL T512,v50,laserON,z0,toolEtna\WObj:=wobjEtna;
    TriggL T513,vl,laserOFF,z0,toolEtna\WObj:=wobjEtna;
    TriggL T514,v50,laserON,z0,toolEtna\WObj:=wobjEtna;
    TriggL T515,vl,laserOFF,z0,toolEtna\WObj:=wobjEtna;
    TriggL T516,v50,laserON,z0,toolEtna\WObj:=wobjEtna;
    TriggL T517,vl,laserOFF,z0,toolEtna\WObj:=wobjEtna;
    TriggL T518,v50,laserON,z0,toolEtna\WObj:=wobjEtna;
    TriggL T519,vl,laserOFF,z0,toolEtna\WObj:=wobjEtna;
    TriggL T520,v50,laserON,z0,toolEtna\WObj:=wobjEtna;
    TriggL T521,vl,laserOFF,z0,toolEtna\WObj:=wobjEtna;
    TriggL T522,v50,laserON,z0,toolEtna\WObj:=wobjEtna;
    TriggL T523,vl,laserOFF,z0,toolEtna\WObj:=wobjEtna;
    TriggL T524,v50,laserON,z0,toolEtna\WObj:=wobjEtna;
    TriggL T525,vl,laserOFF,z0,toolEtna\WObj:=wobjEtna;
    TriggL T526,v50,laserON,z0,toolEtna\WObj:=wobjEtna;
    TriggL T527,vl,laserOFF,z0,toolEtna\WObj:=wobjEtna;
    TriggL T528,v50,laserON,z0,toolEtna\WObj:=wobjEtna;
    TriggL T529,vl,laserOFF,z0,toolEtna\WObj:=wobjEtna;
    TriggL T530,v50,laserON,z0,toolEtna\WObj:=wobjEtna;
    TriggL T531,vl,laserOFF,z0,toolEtna\WObj:=wobjEtna;
    TriggL T532,v50,laserON,z0,toolEtna\WObj:=wobjEtna;
    TriggL T533,vl,laserOFF,z0,toolEtna\WObj:=wobjEtna;
    TriggL T534,v50,laserON,z0,toolEtna\WObj:=wobjEtna;
    TriggL T535,vl,laserOFF,z0,toolEtna\WObj:=wobjEtna;
    TriggL T536,v50,laserON,z0,toolEtna\WObj:=wobjEtna;
    TriggL T537,vl,laserOFF,z0,toolEtna\WObj:=wobjEtna;
    TriggL T538,v50,laserON,z0,toolEtna\WObj:=wobjEtna;
    TriggL T539,vl,laserOFF,z0,toolEtna\WObj:=wobjEtna;
    TriggL T540,v50,laserON,z0,toolEtna\WObj:=wobjEtna;
    TriggL T541,vl,laserOFF,z0,toolEtna\WObj:=wobjEtna;
    TriggL T542,v50,laserON,z0,toolEtna\WObj:=wobjEtna;
    TriggL T543,vl,laserOFF,z0,toolEtna\WObj:=wobjEtna;
    TriggL T544,v50,laserON,z0,toolEtna\WObj:=wobjEtna;
    TriggL T545,vl,laserOFF,z0,toolEtna\WObj:=wobjEtna;
    TriggL T546,v50,laserON,z0,toolEtna\WObj:=wobjEtna;
    TriggL T547,vl,laserOFF,z0,toolEtna\WObj:=wobjEtna;
    TriggL T548,v50,laserON,z0,toolEtna\WObj:=wobjEtna;
    TriggL T549,vl,laserOFF,z0,toolEtna\WObj:=wobjEtna;
    TriggL T550,v50,laserON,z0,toolEtna\WObj:=wobjEtna;
    TriggL T551,vl,laserOFF,z0,toolEtna\WObj:=wobjEtna;
    TriggL T552,v50,laserON,z0,toolEtna\WObj:=wobjEtna;
    TriggL T553,vl,laserOFF,z0,toolEtna\WObj:=wobjEtna;
    TriggL T554,v50,laserON,z0,toolEtna\WObj:=wobjEtna;
    TriggL T555,vl,laserOFF,z0,toolEtna\WObj:=wobjEtna;
    TriggL T556,v50,laserON,z0,toolEtna\WObj:=wobjEtna;
    TriggL T557,vl,laserOFF,z0,toolEtna\WObj:=wobjEtna;
    TriggL T558,v50,laserON,z0,toolEtna\WObj:=wobjEtna;
    TriggL T559,vl,laserOFF,z0,toolEtna\WObj:=wobjEtna;
    TriggL T560,v50,laserON,z0,toolEtna\WObj:=wobjEtna;
    TriggL T561,vl,laserOFF,z0,toolEtna\WObj:=wobjEtna;
    TriggL T562,v50,laserON,z0,toolEtna\WObj:=wobjEtna;
    TriggL T563,vl,laserOFF,z0,toolEtna\WObj:=wobjEtna;
    TriggL T564,v50,laserON,z0,toolEtna\WObj:=wobjEtna;
    TriggL T565,vl,laserOFF,z0,toolEtna\WObj:=wobjEtna;
    TriggL T566,v50,laserON,z0,toolEtna\WObj:=wobjEtna;
    TriggL T567,vl,laserOFF,z0,toolEtna\WObj:=wobjEtna;
    TriggL T568,v50,laserON,z0,toolEtna\WObj:=wobjEtna;
    TriggL T569,vl,laserOFF,z0,toolEtna\WObj:=wobjEtna;
    TriggL T570,v50,laserON,z0,toolEtna\WObj:=wobjEtna;
    TriggL T571,vl,laserOFF,z0,toolEtna\WObj:=wobjEtna;
    TriggL T572,v50,laserON,z0,toolEtna\WObj:=wobjEtna;
    TriggL T573,vl,laserOFF,z0,toolEtna\WObj:=wobjEtna;
    TriggL T574,v50,laserON,z0,toolEtna\WObj:=wobjEtna;
    TriggL T575,vl,laserOFF,z0,toolEtna\WObj:=wobjEtna;
    TriggL T576,v50,laserON,z0,toolEtna\WObj:=wobjEtna;
    TriggL T577,vl,laserOFF,z0,toolEtna\WObj:=wobjEtna;
    TriggL T578,v50,laserON,z0,toolEtna\WObj:=wobjEtna;
    TriggL T579,vl,laserOFF,z0,toolEtna\WObj:=wobjEtna;
    TriggL T580,v50,laserON,z0,toolEtna\WObj:=wobjEtna;
    TriggL T581,vl,laserOFF,z0,toolEtna\WObj:=wobjEtna;
    TriggL T582,v50,laserON,z0,toolEtna\WObj:=wobjEtna;
    TriggL T583,vl,laserOFF,z0,toolEtna\WObj:=wobjEtna;
    TriggL T584,v50,laserON,z0,toolEtna\WObj:=wobjEtna;
    TriggL T585,vl,laserOFF,z0,toolEtna\WObj:=wobjEtna;
    TriggL T586,v50,laserON,z0,toolEtna\WObj:=wobjEtna;
    TriggL T587,vl,laserOFF,z0,toolEtna\WObj:=wobjEtna;
    TriggL T588,v50,laserON,z0,toolEtna\WObj:=wobjEtna;
    TriggL T589,vl,laserOFF,z0,toolEtna\WObj:=wobjEtna;
    TriggL T590,v50,laserON,z0,toolEtna\WObj:=wobjEtna;
    TriggL T591,vl,laserOFF,z0,toolEtna\WObj:=wobjEtna;
    TriggL T592,v50,laserON,z0,toolEtna\WObj:=wobjEtna;
    TriggL T593,vl,laserOFF,z0,toolEtna\WObj:=wobjEtna;
    TriggL T594,v50,laserON,z0,toolEtna\WObj:=wobjEtna;
    TriggL T595,vl,laserOFF,z0,toolEtna\WObj:=wobjEtna;
    TriggL T596,v50,laserON,z0,toolEtna\WObj:=wobjEtna;
    TriggL T597,vl,laserOFF,z0,toolEtna\WObj:=wobjEtna;
    TriggL T598,v50,laserON,z0,toolEtna\WObj:=wobjEtna;
    TriggL T599,vl,laserOFF,z0,toolEtna\WObj:=wobjEtna;
    TriggL T600,v50,laserON,z0,toolEtna\WObj:=wobjEtna;
    TriggL T601,vl,laserOFF,z0,toolEtna\WObj:=wobjEtna;
    TriggL T602,v50,laserON,z0,toolEtna\WObj:=wobjEtna;
    TriggL T603,vl,laserOFF,z0,toolEtna\WObj:=wobjEtna;
    TriggL T604,v50,laserON,z0,toolEtna\WObj:=wobjEtna;
    TriggL T605,vl,laserOFF,z0,toolEtna\WObj:=wobjEtna;
    TriggL T606,v50,laserON,z0,toolEtna\WObj:=wobjEtna;
    TriggL T607,vl,laserOFF,z0,toolEtna\WObj:=wobjEtna;
    TriggL T608,v50,laserON,z0,toolEtna\WObj:=wobjEtna;
    TriggL T609,vl,laserOFF,z0,toolEtna\WObj:=wobjEtna;
    TriggL T610,v50,laserON,z0,toolEtna\WObj:=wobjEtna;
    TriggL T611,vl,laserOFF,z0,toolEtna\WObj:=wobjEtna;
    TriggL T612,v50,laserON,z0,toolEtna\WObj:=wobjEtna;
    TriggL T613,vl,laserOFF,z0,toolEtna\WObj:=wobjEtna;
    TriggL T614,v50,laserON,z0,toolEtna\WObj:=wobjEtna;
    TriggL T615,vl,laserOFF,z0,toolEtna\WObj:=wobjEtna;
    TriggL T616,v50,laserON,z0,toolEtna\WObj:=wobjEtna;
    TriggL T617,vl,laserOFF,z0,toolEtna\WObj:=wobjEtna;
    TriggL T618,v50,laserON,z0,toolEtna\WObj:=wobjEtna;
    TriggL T619,vl,laserOFF,z0,toolEtna\WObj:=wobjEtna;
    TriggL T620,v50,laserON,z0,toolEtna\WObj:=wobjEtna;
    TriggL T621,vl,laserOFF,z0,toolEtna\WObj:=wobjEtna;
    TriggL T622,v50,laserON,z0,toolEtna\WObj:=wobjEtna;
    TriggL T623,vl,laserOFF,z0,toolEtna\WObj:=wobjEtna;
    TriggL T624,v50,laserON,z0,toolEtna\WObj:=wobjEtna;
    TriggL T625,vl,laserOFF,z0,toolEtna\WObj:=wobjEtna;
    TriggL T626,v50,laserON,z0,toolEtna\WObj:=wobjEtna;
    TriggL T627,vl,laserOFF,z0,toolEtna\WObj:=wobjEtna;
    TriggL T628,v50,laserON,z0,toolEtna\WObj:=wobjEtna;
    TriggL T629,vl,laserOFF,z0,toolEtna\WObj:=wobjEtna;
    TriggL T630,v50,laserON,z0,toolEtna\WObj:=wobjEtna;
    TriggL T631,vl,laserOFF,z0,toolEtna\WObj:=wobjEtna;
    TriggL T632,v50,laserON,z0,toolEtna\WObj:=wobjEtna;
    TriggL T633,vl,laserOFF,z0,toolEtna\WObj:=wobjEtna;
    TriggL T634,v50,laserON,z0,toolEtna\WObj:=wobjEtna;
    TriggL T635,vl,laserOFF,z0,toolEtna\WObj:=wobjEtna;
    TriggL T636,v50,laserON,z0,toolEtna\WObj:=wobjEtna;
    TriggL T637,vl,laserOFF,z0,toolEtna\WObj:=wobjEtna;
    TriggL T638,v50,laserON,z0,toolEtna\WObj:=wobjEtna;
    TriggL T639,vl,laserOFF,z0,toolEtna\WObj:=wobjEtna;
    TriggL T640,v50,laserON,z0,toolEtna\WObj:=wobjEtna;
    TriggL T641,vl,laserOFF,z0,toolEtna\WObj:=wobjEtna;
    TriggL T642,v50,laserON,z0,toolEtna\WObj:=wobjEtna;
    TriggL T643,vl,laserOFF,z0,toolEtna\WObj:=wobjEtna;
    TriggL T644,v50,laserON,z0,toolEtna\WObj:=wobjEtna;
    TriggL T645,vl,laserOFF,z0,toolEtna\WObj:=wobjEtna;
    TriggL T646,v50,laserON,z0,toolEtna\WObj:=wobjEtna;
    TriggL T647,vl,laserOFF,z0,toolEtna\WObj:=wobjEtna;
    TriggL T648,v50,laserON,z0,toolEtna\WObj:=wobjEtna;
    TriggL T649,vl,laserOFF,z0,toolEtna\WObj:=wobjEtna;
    TriggL T650,v50,laserON,z0,toolEtna\WObj:=wobjEtna;
    TriggL T651,vl,laserOFF,z0,toolEtna\WObj:=wobjEtna;
    TriggL T652,v50,laserON,z0,toolEtna\WObj:=wobjEtna;
    TriggL T653,vl,laserOFF,z0,toolEtna\WObj:=wobjEtna;
    TriggL T654,v50,laserON,z0,toolEtna\WObj:=wobjEtna;
    TriggL T655,vl,laserOFF,z0,toolEtna\WObj:=wobjEtna;
    TriggL T656,v50,laserON,z0,toolEtna\WObj:=wobjEtna;
    TriggL T657,vl,laserOFF,z0,toolEtna\WObj:=wobjEtna;
    TriggL T658,v50,laserON,z0,toolEtna\WObj:=wobjEtna;
    TriggL T659,vl,laserOFF,z0,toolEtna\WObj:=wobjEtna;
    TriggL T660,v50,laserON,z0,toolEtna\WObj:=wobjEtna;
    TriggL T661,vl,laserOFF,z0,toolEtna\WObj:=wobjEtna;
    TriggL T662,v50,laserON,z0,toolEtna\WObj:=wobjEtna;
    TriggL T663,vl,laserOFF,z0,toolEtna\WObj:=wobjEtna;
    TriggL T664,v50,laserON,z0,toolEtna\WObj:=wobjEtna;
    TriggL T665,vl,laserOFF,z0,toolEtna\WObj:=wobjEtna;
    TriggL T666,v50,laserON,z0,toolEtna\WObj:=wobjEtna;
    TriggL T667,vl,laserOFF,z0,toolEtna\WObj:=wobjEtna;
    TriggL T668,v50,laserON,z0,toolEtna\WObj:=wobjEtna;
    TriggL T669,vl,laserOFF,z0,toolEtna\WObj:=wobjEtna;
    TriggL T670,v50,laserON,z0,toolEtna\WObj:=wobjEtna;
    TriggL T671,vl,laserOFF,z0,toolEtna\WObj:=wobjEtna;
    TriggL T672,v50,laserON,z0,toolEtna\WObj:=wobjEtna;
    TriggL T673,vl,laserOFF,z0,toolEtna\WObj:=wobjEtna;
    TriggL T674,v50,laserON,z0,toolEtna\WObj:=wobjEtna;
    TriggL T675,vl,laserOFF,z0,toolEtna\WObj:=wobjEtna;
    TriggL T676,v50,laserON,z0,toolEtna\WObj:=wobjEtna;
    TriggL T677,vl,laserOFF,z0,toolEtna\WObj:=wobjEtna;
    TriggL T678,v50,laserON,z0,toolEtna\WObj:=wobjEtna;
    TriggL T679,vl,laserOFF,z0,toolEtna\WObj:=wobjEtna;
    TriggL T680,v50,laserON,z0,toolEtna\WObj:=wobjEtna;
    TriggL T681,vl,laserOFF,z0,toolEtna\WObj:=wobjEtna;
    TriggL T682,v50,laserON,z0,toolEtna\WObj:=wobjEtna;
    TriggL T683,vl,laserOFF,z0,toolEtna\WObj:=wobjEtna;
    TriggL T684,v50,laserON,z0,toolEtna\WObj:=wobjEtna;
    TriggL T685,vl,laserOFF,z0,toolEtna\WObj:=wobjEtna;
    TriggL T686,v50,laserON,z0,toolEtna\WObj:=wobjEtna;
    TriggL T687,vl,laserOFF,z0,toolEtna\WObj:=wobjEtna;
    TriggL T688,v50,laserON,z0,toolEtna\WObj:=wobjEtna;
    TriggL T689,vl,laserOFF,z0,toolEtna\WObj:=wobjEtna;
    TriggL T690,v50,laserON,z0,toolEtna\WObj:=wobjEtna;
    TriggL T691,vl,laserOFF,z0,toolEtna\WObj:=wobjEtna;
    TriggL T692,v50,laserON,z0,toolEtna\WObj:=wobjEtna;
    TriggL T693,vl,laserOFF,z0,toolEtna\WObj:=wobjEtna;
    TriggL T694,v50,laserON,z0,toolEtna\WObj:=wobjEtna;
    TriggL T695,vl,laserOFF,z0,toolEtna\WObj:=wobjEtna;
    TriggL T696,v50,laserON,z0,toolEtna\WObj:=wobjEtna;
    TriggL T697,vl,laserOFF,z0,toolEtna\WObj:=wobjEtna;
    TriggL T698,v50,laserON,z0,toolEtna\WObj:=wobjEtna;
    TriggL T699,vl,laserOFF,z0,toolEtna\WObj:=wobjEtna;
    TriggL T700,v50,laserON,z0,toolEtna\WObj:=wobjEtna;
    TriggL T701,vl,laserOFF,z0,toolEtna\WObj:=wobjEtna;
    TriggL T702,v50,laserON,z0,toolEtna\WObj:=wobjEtna;
    TriggL T703,vl,laserOFF,z0,toolEtna\WObj:=wobjEtna;
    TriggL T704,v50,laserON,z0,toolEtna\WObj:=wobjEtna;
    TriggL T705,vl,laserOFF,z0,toolEtna\WObj:=wobjEtna;
    TriggL T706,v50,laserON,z0,toolEtna\WObj:=wobjEtna;
    TriggL T707,vl,laserOFF,z0,toolEtna\WObj:=wobjEtna;
    TriggL T708,v50,laserON,z0,toolEtna\WObj:=wobjEtna;
    TriggL T709,vl,laserOFF,z0,toolEtna\WObj:=wobjEtna;
    TriggL T710,v50,laserON,z0,toolEtna\WObj:=wobjEtna;
    TriggL T711,vl,laserOFF,z0,toolEtna\WObj:=wobjEtna;
    TriggL T712,v50,laserON,z0,toolEtna\WObj:=wobjEtna;
    TriggL T713,vl,laserOFF,z0,toolEtna\WObj:=wobjEtna;
    TriggL T714,v50,laserON,z0,toolEtna\WObj:=wobjEtna;
    TriggL T715,vl,laserOFF,z0,toolEtna\WObj:=wobjEtna;
    TriggL T716,v50,laserON,z0,toolEtna\WObj:=wobjEtna;
    TriggL T717,vl,laserOFF,z0,toolEtna\WObj:=wobjEtna;
    TriggL T718,v50,laserON,z0,toolEtna\WObj:=wobjEtna;
    TriggL T719,vl,laserOFF,z0,toolEtna\WObj:=wobjEtna;
    TriggL T720,v50,laserON,z0,toolEtna\WObj:=wobjEtna;
    TriggL T721,vl,laserOFF,z0,toolEtna\WObj:=wobjEtna;
    TriggL T722,v50,laserON,z0,toolEtna\WObj:=wobjEtna;
    TriggL T723,vl,laserOFF,z0,toolEtna\WObj:=wobjEtna;
    TriggL T724,v50,laserON,z0,toolEtna\WObj:=wobjEtna;
    TriggL T725,vl,laserOFF,z0,toolEtna\WObj:=wobjEtna;
    TriggL T726,v50,laserON,z0,toolEtna\WObj:=wobjEtna;
    TriggL T727,vl,laserOFF,z0,toolEtna\WObj:=wobjEtna;
    TriggL T728,v50,laserON,z0,toolEtna\WObj:=wobjEtna;
    TriggL T729,vl,laserOFF,z0,toolEtna\WObj:=wobjEtna;
    TriggL T730,v50,laserON,z0,toolEtna\WObj:=wobjEtna;
    TriggL T731,vl,laserOFF,z0,toolEtna\WObj:=wobjEtna;
    TriggL T732,v50,laserON,z0,toolEtna\WObj:=wobjEtna;
    TriggL T733,vl,laserOFF,z0,toolEtna\WObj:=wobjEtna;
    TriggL T734,v50,laserON,z0,toolEtna\WObj:=wobjEtna;
    TriggL T735,vl,laserOFF,z0,toolEtna\WObj:=wobjEtna;
    TriggL T736,v50,laserON,z0,toolEtna\WObj:=wobjEtna;
    TriggL T737,vl,laserOFF,z0,toolEtna\WObj:=wobjEtna;
    TriggL T738,v50,laserON,z0,toolEtna\WObj:=wobjEtna;
    TriggL T739,vl,laserOFF,z0,toolEtna\WObj:=wobjEtna;
    TriggL T740,v50,laserON,z0,toolEtna\WObj:=wobjEtna;
    TriggL T741,vl,laserOFF,z0,toolEtna\WObj:=wobjEtna;
    TriggL T742,v50,laserON,z0,toolEtna\WObj:=wobjEtna;
    TriggL T743,vl,laserOFF,z0,toolEtna\WObj:=wobjEtna;
    TriggL T744,v50,laserON,z0,toolEtna\WObj:=wobjEtna;
    TriggL T745,vl,laserOFF,z0,toolEtna\WObj:=wobjEtna;
    TriggL T746,v50,laserON,z0,toolEtna\WObj:=wobjEtna;
    TriggL T747,vl,laserOFF,z0,toolEtna\WObj:=wobjEtna;
    TriggL T748,v50,laserON,z0,toolEtna\WObj:=wobjEtna;
    TriggL T749,vl,laserOFF,z0,toolEtna\WObj:=wobjEtna;
    TriggL T750,v50,laserON,z0,toolEtna\WObj:=wobjEtna;
    TriggL T751,vl,laserOFF,z0,toolEtna\WObj:=wobjEtna;
    TriggL T752,v50,laserON,z0,toolEtna\WObj:=wobjEtna;
    TriggL T753,vl,laserOFF,z0,toolEtna\WObj:=wobjEtna;
    TriggL T754,v50,laserON,z0,toolEtna\WObj:=wobjEtna;
    TriggL T755,vl,laserOFF,z0,toolEtna\WObj:=wobjEtna;
    TriggL T756,v50,laserON,z0,toolEtna\WObj:=wobjEtna;
    TriggL T757,vl,laserOFF,z0,toolEtna\WObj:=wobjEtna;
    TriggL T758,v50,laserON,z0,toolEtna\WObj:=wobjEtna;
    TriggL T759,vl,laserOFF,z0,toolEtna\WObj:=wobjEtna;
    TriggL T760,v50,laserON,z0,toolEtna\WObj:=wobjEtna;
    TriggL T761,vl,laserOFF,z0,toolEtna\WObj:=wobjEtna;
    TriggL T762,v50,laserON,z0,toolEtna\WObj:=wobjEtna;
    TriggL T763,vl,laserOFF,z0,toolEtna\WObj:=wobjEtna;
    TriggL T764,v50,laserON,z0,toolEtna\WObj:=wobjEtna;
    TriggL T765,vl,laserOFF,z0,toolEtna\WObj:=wobjEtna;
    TriggL T766,v50,laserON,z0,toolEtna\WObj:=wobjEtna;
    TriggL T767,vl,laserOFF,z0,toolEtna\WObj:=wobjEtna;
    TriggL T768,v50,laserON,z0,toolEtna\WObj:=wobjEtna;
    TriggL T769,vl,laserOFF,z0,toolEtna\WObj:=wobjEtna;
    TriggL T770,v50,laserON,z0,toolEtna\WObj:=wobjEtna;
    TriggL T771,vl,laserOFF,z0,toolEtna\WObj:=wobjEtna;
    TriggL T772,v50,laserON,z0,toolEtna\WObj:=wobjEtna;
    TriggL T773,vl,laserOFF,z0,toolEtna\WObj:=wobjEtna;
    TriggL T774,v50,laserON,z0,toolEtna\WObj:=wobjEtna;
    TriggL T775,vl,laserOFF,z0,toolEtna\WObj:=wobjEtna;
    TriggL T776,v50,laserON,z0,toolEtna\WObj:=wobjEtna;
    TriggL T777,vl,laserOFF,z0,toolEtna\WObj:=wobjEtna;
    TriggL T778,v50,laserON,z0,toolEtna\WObj:=wobjEtna;
    TriggL T779,vl,laserOFF,z0,toolEtna\WObj:=wobjEtna;
    TriggL T780,v50,laserON,z0,toolEtna\WObj:=wobjEtna;
    TriggL T781,vl,laserOFF,z0,toolEtna\WObj:=wobjEtna;
    TriggL T782,v50,laserON,z0,toolEtna\WObj:=wobjEtna;
    TriggL T783,vl,laserOFF,z0,toolEtna\WObj:=wobjEtna;
    TriggL T784,v50,laserON,z0,toolEtna\WObj:=wobjEtna;
    TriggL T785,vl,laserOFF,z0,toolEtna\WObj:=wobjEtna;
    TriggL T786,v50,laserON,z0,toolEtna\WObj:=wobjEtna;
    TriggL T787,vl,laserOFF,z0,toolEtna\WObj:=wobjEtna;
    TriggL T788,v50,laserON,z0,toolEtna\WObj:=wobjEtna;
    TriggL T789,vl,laserOFF,z0,toolEtna\WObj:=wobjEtna;
    TriggL T790,v50,laserON,z0,toolEtna\WObj:=wobjEtna;
    TriggL T791,vl,laserOFF,z0,toolEtna\WObj:=wobjEtna;
    TriggL T792,v50,laserON,z0,toolEtna\WObj:=wobjEtna;
    TriggL T793,vl,laserOFF,z0,toolEtna\WObj:=wobjEtna;
    TriggL T794,v50,laserON,z0,toolEtna\WObj:=wobjEtna;
    TriggL T795,vl,laserOFF,z0,toolEtna\WObj:=wobjEtna;
    TriggL T796,v50,laserON,z0,toolEtna\WObj:=wobjEtna;
    TriggL T797,vl,laserOFF,z0,toolEtna\WObj:=wobjEtna;
    TriggL T798,v50,laserON,z0,toolEtna\WObj:=wobjEtna;
    TriggL T799,vl,laserOFF,z0,toolEtna\WObj:=wobjEtna;
    TriggL T800,v50,laserON,z0,toolEtna\WObj:=wobjEtna;
    TriggL T801,vl,laserOFF,z0,toolEtna\WObj:=wobjEtna;
    TriggL T802,v50,laserON,z0,toolEtna\WObj:=wobjEtna;
    TriggL T803,vl,laserOFF,z0,toolEtna\WObj:=wobjEtna;
    TriggL T804,v50,laserON,z0,toolEtna\WObj:=wobjEtna;
    TriggL T805,vl,laserOFF,z0,toolEtna\WObj:=wobjEtna;
    TriggL T806,v50,laserON,z0,toolEtna\WObj:=wobjEtna;
    TriggL T807,vl,laserOFF,z0,toolEtna\WObj:=wobjEtna;
    TriggL T808,v50,laserON,z0,toolEtna\WObj:=wobjEtna;
    TriggL T809,vl,laserOFF,z0,toolEtna\WObj:=wobjEtna;
    TriggL T810,v50,laserON,z0,toolEtna\WObj:=wobjEtna;
    TriggL T811,vl,laserOFF,z0,toolEtna\WObj:=wobjEtna;
    TriggL T812,v50,laserON,z0,toolEtna\WObj:=wobjEtna;
    TriggL T813,vl,laserOFF,z0,toolEtna\WObj:=wobjEtna;
    TriggL T814,v50,laserON,z0,toolEtna\WObj:=wobjEtna;
    TriggL T815,vl,laserOFF,z0,toolEtna\WObj:=wobjEtna;
    TriggL T816,v50,laserON,z0,toolEtna\WObj:=wobjEtna;
    TriggL T817,vl,laserOFF,z0,toolEtna\WObj:=wobjEtna;
    TriggL T818,v50,laserON,z0,toolEtna\WObj:=wobjEtna;
    TriggL T819,vl,laserOFF,z0,toolEtna\WObj:=wobjEtna;
    TriggL T820,v50,laserON,z0,toolEtna\WObj:=wobjEtna;
    TriggL T821,vl,laserOFF,z0,toolEtna\WObj:=wobjEtna;
    TriggL T822,v50,laserON,z0,toolEtna\WObj:=wobjEtna;
    TriggL T823,vl,laserOFF,z0,toolEtna\WObj:=wobjEtna;
    TriggL T824,v50,laserON,z0,toolEtna\WObj:=wobjEtna;
    TriggL T825,vl,laserOFF,z0,toolEtna\WObj:=wobjEtna;
    TriggL T826,v50,laserON,z0,toolEtna\WObj:=wobjEtna;
    TriggL T827,vl,laserOFF,z0,toolEtna\WObj:=wobjEtna;
    TriggL T828,v50,laserON,z0,toolEtna\WObj:=wobjEtna;
    TriggL T829,vl,laserOFF,z0,toolEtna\WObj:=wobjEtna;
    TriggL T830,v50,laserON,z0,toolEtna\WObj:=wobjEtna;
    TriggL T831,vl,laserOFF,z0,toolEtna\WObj:=wobjEtna;
    TriggL T832,v50,laserON,z0,toolEtna\WObj:=wobjEtna;
    TriggL T833,vl,laserOFF,z0,toolEtna\WObj:=wobjEtna;
    TriggL T834,v50,laserON,z0,toolEtna\WObj:=wobjEtna;
    TriggL T835,vl,laserOFF,z0,toolEtna\WObj:=wobjEtna;
    TriggL T836,v50,laserON,z0,toolEtna\WObj:=wobjEtna;
    TriggL T837,vl,laserOFF,z0,toolEtna\WObj:=wobjEtna;
    TriggL T838,v50,laserON,z0,toolEtna\WObj:=wobjEtna;
    TriggL T839,vl,laserOFF,z0,toolEtna\WObj:=wobjEtna;
    TriggL T840,v50,laserON,z0,toolEtna\WObj:=wobjEtna;
    TriggL T841,vl,laserOFF,z0,toolEtna\WObj:=wobjEtna;
    TriggL T842,v50,laserON,z0,toolEtna\WObj:=wobjEtna;
    TriggL T843,vl,laserOFF,z0,toolEtna\WObj:=wobjEtna;
    TriggL T844,v50,laserON,z0,toolEtna\WObj:=wobjEtna;
    TriggL T845,vl,laserOFF,z0,toolEtna\WObj:=wobjEtna;
    TriggL T846,v50,laserON,z0,toolEtna\WObj:=wobjEtna;
    TriggL T847,vl,laserOFF,z0,toolEtna\WObj:=wobjEtna;
    TriggL T848,v50,laserON,z0,toolEtna\WObj:=wobjEtna;
    TriggL T849,vl,laserOFF,z0,toolEtna\WObj:=wobjEtna;
    TriggL T850,v50,laserON,z0,toolEtna\WObj:=wobjEtna;
    TriggL T851,vl,laserOFF,z0,toolEtna\WObj:=wobjEtna;
    TriggL T852,v50,laserON,z0,toolEtna\WObj:=wobjEtna;
    TriggL T853,vl,laserOFF,z0,toolEtna\WObj:=wobjEtna;
    TriggL T854,v50,laserON,z0,toolEtna\WObj:=wobjEtna;
    TriggL T855,vl,laserOFF,z0,toolEtna\WObj:=wobjEtna;
    TriggL T856,v50,laserON,z0,toolEtna\WObj:=wobjEtna;
    TriggL T857,vl,laserOFF,z0,toolEtna\WObj:=wobjEtna;
    TriggL T858,v50,laserON,z0,toolEtna\WObj:=wobjEtna;
    TriggL T859,vl,laserOFF,z0,toolEtna\WObj:=wobjEtna;
    TriggL T860,v50,laserON,z0,toolEtna\WObj:=wobjEtna;
    TriggL T861,vl,laserOFF,z0,toolEtna\WObj:=wobjEtna;
    TriggL T862,v50,laserON,z0,toolEtna\WObj:=wobjEtna;
    TriggL T863,vl,laserOFF,z0,toolEtna\WObj:=wobjEtna;
    TriggL T864,v50,laserON,z0,toolEtna\WObj:=wobjEtna;
    TriggL T865,vl,laserOFF,z0,toolEtna\WObj:=wobjEtna;
    TriggL T866,v50,laserON,z0,toolEtna\WObj:=wobjEtna;
    TriggL T867,vl,laserOFF,z0,toolEtna\WObj:=wobjEtna;
    TriggL T868,v50,laserON,z0,toolEtna\WObj:=wobjEtna;
    TriggL T869,vl,laserOFF,z0,toolEtna\WObj:=wobjEtna;
    TriggL T870,v50,laserON,z0,toolEtna\WObj:=wobjEtna;
    TriggL T871,vl,laserOFF,z0,toolEtna\WObj:=wobjEtna;
    TriggL T872,v50,laserON,z0,toolEtna\WObj:=wobjEtna;
    TriggL T873,vl,laserOFF,z0,toolEtna\WObj:=wobjEtna;
    TriggL T874,v50,laserON,z0,toolEtna\WObj:=wobjEtna;
    TriggL T875,vl,laserOFF,z0,toolEtna\WObj:=wobjEtna;
    TriggL T876,v50,laserON,z0,toolEtna\WObj:=wobjEtna;
    TriggL T877,vl,laserOFF,z0,toolEtna\WObj:=wobjEtna;
    TriggL T878,v50,laserON,z0,toolEtna\WObj:=wobjEtna;
    TriggL T879,vl,laserOFF,z0,toolEtna\WObj:=wobjEtna;
    TriggL T880,v50,laserON,z0,toolEtna\WObj:=wobjEtna;
    TriggL T881,vl,laserOFF,z0,toolEtna\WObj:=wobjEtna;
    TriggL T882,v50,laserON,z0,toolEtna\WObj:=wobjEtna;
    TriggL T883,vl,laserOFF,z0,toolEtna\WObj:=wobjEtna;
    TriggL T884,v50,laserON,z0,toolEtna\WObj:=wobjEtna;
    TriggL T885,vl,laserOFF,z0,toolEtna\WObj:=wobjEtna;
    TriggL T886,v50,laserON,z0,toolEtna\WObj:=wobjEtna;
    TriggL T887,vl,laserOFF,z0,toolEtna\WObj:=wobjEtna;
    TriggL T888,v50,laserON,z0,toolEtna\WObj:=wobjEtna;
    TriggL T889,vl,laserOFF,z0,toolEtna\WObj:=wobjEtna;
    TriggL T890,v50,laserON,z0,toolEtna\WObj:=wobjEtna;
    TriggL T891,vl,laserOFF,z0,toolEtna\WObj:=wobjEtna;
    TriggL T892,v50,laserON,z0,toolEtna\WObj:=wobjEtna;
    TriggL T893,vl,laserOFF,z0,toolEtna\WObj:=wobjEtna;
    TriggL T894,v50,laserON,z0,toolEtna\WObj:=wobjEtna;
    TriggL T895,vl,laserOFF,z0,toolEtna\WObj:=wobjEtna;
    TriggL T896,v50,laserON,z0,toolEtna\WObj:=wobjEtna;
    TriggL T897,vl,laserOFF,z0,toolEtna\WObj:=wobjEtna;
    TriggL T898,v50,laserON,z0,toolEtna\WObj:=wobjEtna;
    TriggL T899,vl,laserOFF,z0,toolEtna\WObj:=wobjEtna;
    TriggL T900,v50,laserON,z0,toolEtna\WObj:=wobjEtna;
    TriggL T901,vl,laserOFF,z0,toolEtna\WObj:=wobjEtna;
    TriggL T902,v50,laserON,z0,toolEtna\WObj:=wobjEtna;
    TriggL T903,vl,laserOFF,z0,toolEtna\WObj:=wobjEtna;
    TriggL T904,v50,laserON,z0,toolEtna\WObj:=wobjEtna;
    TriggL T905,vl,laserOFF,z0,toolEtna\WObj:=wobjEtna;
    TriggL T906,v50,laserON,z0,toolEtna\WObj:=wobjEtna;
    TriggL T907,vl,laserOFF,z0,toolEtna\WObj:=wobjEtna;
    TriggL T908,v50,laserON,z0,toolEtna\WObj:=wobjEtna;
    TriggL T909,vl,laserOFF,z0,toolEtna\WObj:=wobjEtna;
    TriggL T910,v50,laserON,z0,toolEtna\WObj:=wobjEtna;
    TriggL T911,vl,laserOFF,z0,toolEtna\WObj:=wobjEtna;
    TriggL T912,v50,laserON,z0,toolEtna\WObj:=wobjEtna;
    TriggL T913,vl,laserOFF,z0,toolEtna\WObj:=wobjEtna;
    TriggL T914,v50,laserON,z0,toolEtna\WObj:=wobjEtna;
    TriggL T915,vl,laserOFF,z0,toolEtna\WObj:=wobjEtna;
    TriggL T916,v50,laserON,z0,toolEtna\WObj:=wobjEtna;
    TriggL T917,vl,laserOFF,z0,toolEtna\WObj:=wobjEtna;
    TriggL T918,v50,laserON,z0,toolEtna\WObj:=wobjEtna;
    TriggL T919,vl,laserOFF,z0,toolEtna\WObj:=wobjEtna;
    TriggL T920,v50,laserON,z0,toolEtna\WObj:=wobjEtna;
    TriggL T921,vl,laserOFF,z0,toolEtna\WObj:=wobjEtna;
    TriggL T922,v50,laserON,z0,toolEtna\WObj:=wobjEtna;
    TriggL T923,vl,laserOFF,z0,toolEtna\WObj:=wobjEtna;
    TriggL T924,v50,laserON,z0,toolEtna\WObj:=wobjEtna;
    TriggL T925,vl,laserOFF,z0,toolEtna\WObj:=wobjEtna;
    TriggL T926,v50,laserON,z0,toolEtna\WObj:=wobjEtna;
    TriggL T927,vl,laserOFF,z0,toolEtna\WObj:=wobjEtna;
    TriggL T928,v50,laserON,z0,toolEtna\WObj:=wobjEtna;
    TriggL T929,vl,laserOFF,z0,toolEtna\WObj:=wobjEtna;
    TriggL T930,v50,laserON,z0,toolEtna\WObj:=wobjEtna;
    TriggL T931,vl,laserOFF,z0,toolEtna\WObj:=wobjEtna;
    TriggL T932,v50,laserON,z0,toolEtna\WObj:=wobjEtna;
    TriggL T933,vl,laserOFF,z0,toolEtna\WObj:=wobjEtna;
    TriggL T934,v50,laserON,z0,toolEtna\WObj:=wobjEtna;
    TriggL T935,vl,laserOFF,z0,toolEtna\WObj:=wobjEtna;
    TriggL T936,v50,laserON,z0,toolEtna\WObj:=wobjEtna;
    TriggL T937,vl,laserOFF,z0,toolEtna\WObj:=wobjEtna;
    TriggL T938,v50,laserON,z0,toolEtna\WObj:=wobjEtna;
    TriggL T939,vl,laserOFF,z0,toolEtna\WObj:=wobjEtna;
    TriggL T940,v50,laserON,z0,toolEtna\WObj:=wobjEtna;
    TriggL T941,vl,laserOFF,z0,toolEtna\WObj:=wobjEtna;
    TriggL T942,v50,laserON,z0,toolEtna\WObj:=wobjEtna;
    TriggL T943,vl,laserOFF,z0,toolEtna\WObj:=wobjEtna;
    TriggL T944,v50,laserON,z0,toolEtna\WObj:=wobjEtna;
    TriggL T945,vl,laserOFF,z0,toolEtna\WObj:=wobjEtna;
    TriggL T946,v50,laserON,z0,toolEtna\WObj:=wobjEtna;
    TriggL T947,vl,laserOFF,z0,toolEtna\WObj:=wobjEtna;
    TriggL T948,v50,laserON,z0,toolEtna\WObj:=wobjEtna;
    TriggL T949,vl,laserOFF,z0,toolEtna\WObj:=wobjEtna;
    TriggL T950,v50,laserON,z0,toolEtna\WObj:=wobjEtna;
    TriggL T951,vl,laserOFF,z0,toolEtna\WObj:=wobjEtna;
    TriggL T952,v50,laserON,z0,toolEtna\WObj:=wobjEtna;
    TriggL T953,vl,laserOFF,z0,toolEtna\WObj:=wobjEtna;
    TriggL T954,v50,laserON,z0,toolEtna\WObj:=wobjEtna;
    TriggL T955,vl,laserOFF,z0,toolEtna\WObj:=wobjEtna;
    TriggL T956,v50,laserON,z0,toolEtna\WObj:=wobjEtna;
    TriggL T957,vl,laserOFF,z0,toolEtna\WObj:=wobjEtna;
    TriggL T958,v50,laserON,z0,toolEtna\WObj:=wobjEtna;
    TriggL T959,vl,laserOFF,z0,toolEtna\WObj:=wobjEtna;
    TriggL T960,v50,laserON,z0,toolEtna\WObj:=wobjEtna;
    TriggL T961,vl,laserOFF,z0,toolEtna\WObj:=wobjEtna;
    TriggL T962,v50,laserON,z0,toolEtna\WObj:=wobjEtna;
    TriggL T963,vl,laserOFF,z0,toolEtna\WObj:=wobjEtna;
    TriggL T964,v50,laserON,z0,toolEtna\WObj:=wobjEtna;
    TriggL T965,vl,laserOFF,z0,toolEtna\WObj:=wobjEtna;
    TriggL T966,v50,laserON,z0,toolEtna\WObj:=wobjEtna;
    TriggL T967,vl,laserOFF,z0,toolEtna\WObj:=wobjEtna;
    TriggL T968,v50,laserON,z0,toolEtna\WObj:=wobjEtna;
    TriggL T969,vl,laserOFF,z0,toolEtna\WObj:=wobjEtna;
    TriggL T970,v50,laserON,z0,toolEtna\WObj:=wobjEtna;
    TriggL T971,vl,laserOFF,z0,toolEtna\WObj:=wobjEtna;
    TriggL T972,v50,laserON,z0,toolEtna\WObj:=wobjEtna;
    TriggL T973,vl,laserOFF,z0,toolEtna\WObj:=wobjEtna;
    TriggL T974,v50,laserON,z0,toolEtna\WObj:=wobjEtna;
    TriggL T975,vl,laserOFF,z0,toolEtna\WObj:=wobjEtna;
    TriggL T976,v50,laserON,z0,toolEtna\WObj:=wobjEtna;
    TriggL T977,vl,laserOFF,z0,toolEtna\WObj:=wobjEtna;
    TriggL T978,v50,laserON,z0,toolEtna\WObj:=wobjEtna;
    TriggL T979,vl,laserOFF,z0,toolEtna\WObj:=wobjEtna;
    TriggL T980,v50,laserON,z0,toolEtna\WObj:=wobjEtna;
    TriggL T981,vl,laserOFF,z0,toolEtna\WObj:=wobjEtna;
    TriggL T982,v50,laserON,z0,toolEtna\WObj:=wobjEtna;
    TriggL T983,vl,laserOFF,z0,toolEtna\WObj:=wobjEtna;
    TriggL T984,v50,laserON,z0,toolEtna\WObj:=wobjEtna;
    TriggL T985,vl,laserOFF,z0,toolEtna\WObj:=wobjEtna;
    TriggL T986,v50,laserON,z0,toolEtna\WObj:=wobjEtna;
    TriggL T987,vl,laserOFF,z0,toolEtna\WObj:=wobjEtna;
    TriggL T988,v50,laserON,z0,toolEtna\WObj:=wobjEtna;
    TriggL T989,vl,laserOFF,z0,toolEtna\WObj:=wobjEtna;
    TriggL T990,v50,laserON,z0,toolEtna\WObj:=wobjEtna;
    TriggL T991,vl,laserOFF,z0,toolEtna\WObj:=wobjEtna;
    TriggL T992,v50,laserON,z0,toolEtna\WObj:=wobjEtna;
    TriggL T993,vl,laserOFF,z0,toolEtna\WObj:=wobjEtna;
    TriggL T994,v50,laserON,z0,toolEtna\WObj:=wobjEtna;
    TriggL T995,vl,laserOFF,z0,toolEtna\WObj:=wobjEtna;
    TriggL T996,v50,laserON,z0,toolEtna\WObj:=wobjEtna;
    TriggL T997,vl,laserOFF,z0,toolEtna\WObj:=wobjEtna;
    TriggL T998,v50,laserON,z0,toolEtna\WObj:=wobjEtna;
    TriggL T999,vl,laserOFF,z0,toolEtna\WObj:=wobjEtna;
    TriggL T1000,v50,laserON,z0,toolEtna\WObj:=wobjEtna;
    TriggL T1001,vl,laserOFF,z0,toolEtna\WObj:=wobjEtna;
    TriggL T1002,v50,laserON,z0,toolEtna\WObj:=wobjEtna;
    TriggL T1003,vl,laserOFF,z0,toolEtna\WObj:=wobjEtna;
    TriggL T1004,v50,laserON,z0,toolEtna\WObj:=wobjEtna;
    TriggL T1005,vl,laserOFF,z0,toolEtna\WObj:=wobjEtna;
    TriggL T1006,v50,laserON,z0,toolEtna\WObj:=wobjEtna;
    TriggL T1007,vl,laserOFF,z0,toolEtna\WObj:=wobjEtna;
    TriggL T1008,v50,laserON,z0,toolEtna\WObj:=wobjEtna;
    TriggL T1009,vl,laserOFF,z0,toolEtna\WObj:=wobjEtna;
    TriggL T1010,v50,laserON,z0,toolEtna\WObj:=wobjEtna;
    TriggL T1011,vl,laserOFF,z0,toolEtna\WObj:=wobjEtna;
    TriggL T1012,v50,laserON,z0,toolEtna\WObj:=wobjEtna;
    TriggL T1013,vl,laserOFF,z0,toolEtna\WObj:=wobjEtna;
    TriggL T1014,v50,laserON,z0,toolEtna\WObj:=wobjEtna;
    TriggL T1015,vl,laserOFF,z0,toolEtna\WObj:=wobjEtna;
    TriggL T1016,v50,laserON,z0,toolEtna\WObj:=wobjEtna;
    TriggL T1017,vl,laserOFF,z0,toolEtna\WObj:=wobjEtna;
    TriggL T1018,v50,laserON,z0,toolEtna\WObj:=wobjEtna;
    TriggL T1019,vl,laserOFF,z0,toolEtna\WObj:=wobjEtna;
    TriggL T1020,v50,laserON,z0,toolEtna\WObj:=wobjEtna;
    TriggL T1021,vl,laserOFF,z0,toolEtna\WObj:=wobjEtna;
    TriggL T1022,v50,laserON,z0,toolEtna\WObj:=wobjEtna;
    TriggL T1023,vl,laserOFF,z0,toolEtna\WObj:=wobjEtna;
    TriggL T1024,v50,laserON,z0,toolEtna\WObj:=wobjEtna;
    TriggL T1025,vl,laserOFF,z0,toolEtna\WObj:=wobjEtna;
    TriggL T1026,v50,laserON,z0,toolEtna\WObj:=wobjEtna;
    TriggL T1027,vl,laserOFF,z0,toolEtna\WObj:=wobjEtna;
    TriggL T1028,v50,laserON,z0,toolEtna\WObj:=wobjEtna;
    TriggL T1029,vl,laserOFF,z0,toolEtna\WObj:=wobjEtna;
    TriggL T1030,v50,laserON,z0,toolEtna\WObj:=wobjEtna;
    TriggL T1031,vl,laserOFF,z0,toolEtna\WObj:=wobjEtna;
    TriggL T1032,v50,laserON,z0,toolEtna\WObj:=wobjEtna;
    TriggL T1033,vl,laserOFF,z0,toolEtna\WObj:=wobjEtna;
    TriggL T1034,v50,laserON,z0,toolEtna\WObj:=wobjEtna;
    TriggL T1035,vl,laserOFF,z0,toolEtna\WObj:=wobjEtna;
    TriggL T1036,v50,laserON,z0,toolEtna\WObj:=wobjEtna;
    TriggL T1037,vl,laserOFF,z0,toolEtna\WObj:=wobjEtna;
    TriggL T1038,v50,laserON,z0,toolEtna\WObj:=wobjEtna;
    TriggL T1039,vl,laserOFF,z0,toolEtna\WObj:=wobjEtna;
    TriggL T1040,v50,laserON,z0,toolEtna\WObj:=wobjEtna;
    TriggL T1041,vl,laserOFF,z0,toolEtna\WObj:=wobjEtna;
    TriggL T1042,v50,laserON,z0,toolEtna\WObj:=wobjEtna;
    TriggL T1043,vl,laserOFF,z0,toolEtna\WObj:=wobjEtna;
    TriggL T1044,v50,laserON,z0,toolEtna\WObj:=wobjEtna;
    TriggL T1045,vl,laserOFF,z0,toolEtna\WObj:=wobjEtna;
    TriggL T1046,v50,laserON,z0,toolEtna\WObj:=wobjEtna;
    TriggL T1047,vl,laserOFF,z0,toolEtna\WObj:=wobjEtna;
    TriggL T1048,v50,laserON,z0,toolEtna\WObj:=wobjEtna;
    TriggL T1049,vl,laserOFF,z0,toolEtna\WObj:=wobjEtna;
    TriggL T1050,v50,laserON,z0,toolEtna\WObj:=wobjEtna;
    TriggL T1051,vl,laserOFF,z0,toolEtna\WObj:=wobjEtna;
    TriggL T1052,v50,laserON,z0,toolEtna\WObj:=wobjEtna;
    TriggL T1053,vl,laserOFF,z0,toolEtna\WObj:=wobjEtna;
    TriggL T1054,v50,laserON,z0,toolEtna\WObj:=wobjEtna;
    TriggL T1055,vl,laserOFF,z0,toolEtna\WObj:=wobjEtna;
    TriggL T1056,v50,laserON,z0,toolEtna\WObj:=wobjEtna;
    TriggL T1057,vl,laserOFF,z0,toolEtna\WObj:=wobjEtna;
    TriggL T1058,v50,laserON,z0,toolEtna\WObj:=wobjEtna;
    TriggL T1059,vl,laserOFF,z0,toolEtna\WObj:=wobjEtna;
    TriggL T1060,v50,laserON,z0,toolEtna\WObj:=wobjEtna;
    TriggL T1061,vl,laserOFF,z0,toolEtna\WObj:=wobjEtna;
    TriggL T1062,v50,laserON,z0,toolEtna\WObj:=wobjEtna;
    TriggL T1063,vl,laserOFF,z0,toolEtna\WObj:=wobjEtna;
    TriggL T1064,v50,laserON,z0,toolEtna\WObj:=wobjEtna;
    TriggL T1065,vl,laserOFF,z0,toolEtna\WObj:=wobjEtna;
    TriggL T1066,v50,laserON,z0,toolEtna\WObj:=wobjEtna;
    TriggL T1067,vl,laserOFF,z0,toolEtna\WObj:=wobjEtna;
    TriggL T1068,v50,laserON,z0,toolEtna\WObj:=wobjEtna;
    TriggL T1069,vl,laserOFF,z0,toolEtna\WObj:=wobjEtna;
    TriggL T1070,v50,laserON,z0,toolEtna\WObj:=wobjEtna;
    TriggL T1071,vl,laserOFF,z0,toolEtna\WObj:=wobjEtna;
    TriggL T1072,v50,laserON,z0,toolEtna\WObj:=wobjEtna;
    TriggL T1073,vl,laserOFF,z0,toolEtna\WObj:=wobjEtna;
    TriggL T1074,v50,laserON,z0,toolEtna\WObj:=wobjEtna;
    TriggL T1075,vl,laserOFF,z0,toolEtna\WObj:=wobjEtna;
    TriggL T1076,v50,laserON,z0,toolEtna\WObj:=wobjEtna;
    TriggL T1077,vl,laserOFF,z0,toolEtna\WObj:=wobjEtna;
    TriggL T1078,v50,laserON,z0,toolEtna\WObj:=wobjEtna;
    TriggL T1079,vl,laserOFF,z0,toolEtna\WObj:=wobjEtna;
    TriggL T1080,v50,laserON,z0,toolEtna\WObj:=wobjEtna;
    TriggL T1081,vl,laserOFF,z0,toolEtna\WObj:=wobjEtna;
    TriggL T1082,v50,laserON,z0,toolEtna\WObj:=wobjEtna;
    TriggL T1083,vl,laserOFF,z0,toolEtna\WObj:=wobjEtna;
    TriggL T1084,v50,laserON,z0,toolEtna\WObj:=wobjEtna;
    TriggL T1085,vl,laserOFF,z0,toolEtna\WObj:=wobjEtna;
    TriggL T1086,v50,laserON,z0,toolEtna\WObj:=wobjEtna;
    TriggL T1087,vl,laserOFF,z0,toolEtna\WObj:=wobjEtna;
    TriggL T1088,v50,laserON,z0,toolEtna\WObj:=wobjEtna;
    TriggL T1089,vl,laserOFF,z0,toolEtna\WObj:=wobjEtna;
    TriggL T1090,v50,laserON,z0,toolEtna\WObj:=wobjEtna;
    TriggL T1091,vl,laserOFF,z0,toolEtna\WObj:=wobjEtna;
    TriggL T1092,v50,laserON,z0,toolEtna\WObj:=wobjEtna;
    TriggL T1093,vl,laserOFF,z0,toolEtna\WObj:=wobjEtna;
    TriggL T1094,v50,laserON,z0,toolEtna\WObj:=wobjEtna;
    TriggL T1095,vl,laserOFF,z0,toolEtna\WObj:=wobjEtna;
    TriggL T1096,v50,laserON,z0,toolEtna\WObj:=wobjEtna;
    TriggL T1097,vl,laserOFF,z0,toolEtna\WObj:=wobjEtna;
    TriggL T1098,v50,laserON,z0,toolEtna\WObj:=wobjEtna;
    TriggL T1099,vl,laserOFF,z0,toolEtna\WObj:=wobjEtna;
    TriggL T1100,v50,laserON,z0,toolEtna\WObj:=wobjEtna;
    TriggL T1101,vl,laserOFF,z0,toolEtna\WObj:=wobjEtna;
    TriggL T1102,v50,laserON,z0,toolEtna\WObj:=wobjEtna;
    TriggL T1103,vl,laserOFF,z0,toolEtna\WObj:=wobjEtna;
    TriggL T1104,v50,laserON,z0,toolEtna\WObj:=wobjEtna;
    TriggL T1105,vl,laserOFF,z0,toolEtna\WObj:=wobjEtna;
    TriggL T1106,v50,laserON,z0,toolEtna\WObj:=wobjEtna;
    TriggL T1107,vl,laserOFF,z0,toolEtna\WObj:=wobjEtna;
    TriggL T1108,v50,laserON,z0,toolEtna\WObj:=wobjEtna;
    TriggL T1109,vl,laserOFF,z0,toolEtna\WObj:=wobjEtna;
    TriggL T1110,v50,laserON,z0,toolEtna\WObj:=wobjEtna;
    TriggL T1111,vl,laserOFF,z0,toolEtna\WObj:=wobjEtna;
    TriggL T1112,v50,laserON,z0,toolEtna\WObj:=wobjEtna;
    TriggL T1113,vl,laserOFF,z0,toolEtna\WObj:=wobjEtna;
    TriggL T1114,v50,laserON,z0,toolEtna\WObj:=wobjEtna;
    TriggL T1115,vl,laserOFF,z0,toolEtna\WObj:=wobjEtna;
    TriggL T1116,v50,laserON,z0,toolEtna\WObj:=wobjEtna;
    TriggL T1117,vl,laserOFF,z0,toolEtna\WObj:=wobjEtna;
    TriggL T1118,v50,laserON,z0,toolEtna\WObj:=wobjEtna;
    TriggL T1119,vl,laserOFF,z0,toolEtna\WObj:=wobjEtna;
    TriggL T1120,v50,laserON,z0,toolEtna\WObj:=wobjEtna;
    TriggL T1121,vl,laserOFF,z0,toolEtna\WObj:=wobjEtna;
    TriggL T1122,v50,laserON,z0,toolEtna\WObj:=wobjEtna;
    TriggL T1123,vl,laserOFF,z0,toolEtna\WObj:=wobjEtna;
    TriggL T1124,v50,laserON,z0,toolEtna\WObj:=wobjEtna;
    TriggL T1125,vl,laserOFF,z0,toolEtna\WObj:=wobjEtna;
    TriggL T1126,v50,laserON,z0,toolEtna\WObj:=wobjEtna;
    TriggL T1127,vl,laserOFF,z0,toolEtna\WObj:=wobjEtna;
    TriggL T1128,v50,laserON,z0,toolEtna\WObj:=wobjEtna;
    TriggL T1129,vl,laserOFF,z0,toolEtna\WObj:=wobjEtna;
    TriggL T1130,v50,laserON,z0,toolEtna\WObj:=wobjEtna;
    TriggL T1131,vl,laserOFF,z0,toolEtna\WObj:=wobjEtna;
    TriggL T1132,v50,laserON,z0,toolEtna\WObj:=wobjEtna;
    TriggL T1133,vl,laserOFF,z0,toolEtna\WObj:=wobjEtna;
    TriggL T1134,v50,laserON,z0,toolEtna\WObj:=wobjEtna;
    TriggL T1135,vl,laserOFF,z0,toolEtna\WObj:=wobjEtna;
    TriggL T1136,v50,laserON,z0,toolEtna\WObj:=wobjEtna;
    TriggL T1137,vl,laserOFF,z0,toolEtna\WObj:=wobjEtna;
    TriggL T1138,v50,laserON,z0,toolEtna\WObj:=wobjEtna;
    TriggL T1139,vl,laserOFF,z0,toolEtna\WObj:=wobjEtna;
    TriggL T1140,v50,laserON,z0,toolEtna\WObj:=wobjEtna;
    TriggL T1141,vl,laserOFF,z0,toolEtna\WObj:=wobjEtna;
    TriggL T1142,v50,laserON,z0,toolEtna\WObj:=wobjEtna;
    TriggL T1143,vl,laserOFF,z0,toolEtna\WObj:=wobjEtna;
    TriggL T1144,v50,laserON,z0,toolEtna\WObj:=wobjEtna;
    TriggL T1145,vl,laserOFF,z0,toolEtna\WObj:=wobjEtna;
    TriggL T1146,v50,laserON,z0,toolEtna\WObj:=wobjEtna;
    TriggL T1147,vl,laserOFF,z0,toolEtna\WObj:=wobjEtna;
    TriggL T1148,v50,laserON,z0,toolEtna\WObj:=wobjEtna;
    TriggL T1149,vl,laserOFF,z0,toolEtna\WObj:=wobjEtna;
    TriggL T1150,v50,laserON,z0,toolEtna\WObj:=wobjEtna;
    TriggL T1151,vl,laserOFF,z0,toolEtna\WObj:=wobjEtna;
    TriggL T1152,v50,laserON,z0,toolEtna\WObj:=wobjEtna;
    TriggL T1153,vl,laserOFF,z0,toolEtna\WObj:=wobjEtna;
    TriggL T1154,v50,laserON,z0,toolEtna\WObj:=wobjEtna;
    TriggL T1155,vl,laserOFF,z0,toolEtna\WObj:=wobjEtna;
    TriggL T1156,v50,laserON,z0,toolEtna\WObj:=wobjEtna;
    TriggL T1157,vl,laserOFF,z0,toolEtna\WObj:=wobjEtna;
    TriggL T1158,v50,laserON,z0,toolEtna\WObj:=wobjEtna;
    TriggL T1159,vl,laserOFF,z0,toolEtna\WObj:=wobjEtna;
    TriggL T1160,v50,laserON,z0,toolEtna\WObj:=wobjEtna;
    TriggL T1161,vl,laserOFF,z0,toolEtna\WObj:=wobjEtna;
    TriggL T1162,v50,laserON,z0,toolEtna\WObj:=wobjEtna;
    TriggL T1163,vl,laserOFF,z0,toolEtna\WObj:=wobjEtna;
    TriggL T1164,v50,laserON,z0,toolEtna\WObj:=wobjEtna;
    TriggL T1165,vl,laserOFF,z0,toolEtna\WObj:=wobjEtna;
    TriggL T1166,v50,laserON,z0,toolEtna\WObj:=wobjEtna;
    TriggL T1167,vl,laserOFF,z0,toolEtna\WObj:=wobjEtna;
    TriggL T1168,v50,laserON,z0,toolEtna\WObj:=wobjEtna;
    TriggL T1169,vl,laserOFF,z0,toolEtna\WObj:=wobjEtna;
    TriggL T1170,v50,laserON,z0,toolEtna\WObj:=wobjEtna;
    TriggL T1171,vl,laserOFF,z0,toolEtna\WObj:=wobjEtna;
    TriggL T1172,v50,laserON,z0,toolEtna\WObj:=wobjEtna;
    TriggL T1173,vl,laserOFF,z0,toolEtna\WObj:=wobjEtna;
    TriggL T1174,v50,laserON,z0,toolEtna\WObj:=wobjEtna;
    TriggL T1175,vl,laserOFF,z0,toolEtna\WObj:=wobjEtna;
    TriggL T1176,v50,laserON,z0,toolEtna\WObj:=wobjEtna;
    TriggL T1177,vl,laserOFF,z0,toolEtna\WObj:=wobjEtna;
    TriggL T1178,v50,laserON,z0,toolEtna\WObj:=wobjEtna;
    TriggL T1179,vl,laserOFF,z0,toolEtna\WObj:=wobjEtna;
    TriggL T1180,v50,laserON,z0,toolEtna\WObj:=wobjEtna;
    TriggL T1181,vl,laserOFF,z0,toolEtna\WObj:=wobjEtna;
    TriggL T1182,v50,laserON,z0,toolEtna\WObj:=wobjEtna;
    TriggL T1183,vl,laserOFF,z0,toolEtna\WObj:=wobjEtna;
    TriggL T1184,v50,laserON,z0,toolEtna\WObj:=wobjEtna;
    TriggL T1185,vl,laserOFF,z0,toolEtna\WObj:=wobjEtna;
    TriggL T1186,v50,laserON,z0,toolEtna\WObj:=wobjEtna;
    TriggL T1187,vl,laserOFF,z0,toolEtna\WObj:=wobjEtna;
    TriggL T1188,v50,laserON,z0,toolEtna\WObj:=wobjEtna;
    TriggL T1189,vl,laserOFF,z0,toolEtna\WObj:=wobjEtna;
    TriggL T1190,v50,laserON,z0,toolEtna\WObj:=wobjEtna;
    TriggL T1191,vl,laserOFF,z0,toolEtna\WObj:=wobjEtna;
    TriggL T1192,v50,laserON,z0,toolEtna\WObj:=wobjEtna;
    TriggL T1193,vl,laserOFF,z0,toolEtna\WObj:=wobjEtna;
    TriggL T1194,v50,laserON,z0,toolEtna\WObj:=wobjEtna;
    TriggL T1195,vl,laserOFF,z0,toolEtna\WObj:=wobjEtna;
    TriggL T1196,v50,laserON,z0,toolEtna\WObj:=wobjEtna;
    TriggL T1197,vl,laserOFF,z0,toolEtna\WObj:=wobjEtna;
    TriggL T1198,v50,laserON,z0,toolEtna\WObj:=wobjEtna;
    TriggL T1199,vl,laserOFF,z0,toolEtna\WObj:=wobjEtna;
    TriggL T1200,v50,laserON,z0,toolEtna\WObj:=wobjEtna;
    TriggL T1201,vl,laserOFF,z0,toolEtna\WObj:=wobjEtna;
    TriggL T1202,v50,laserON,z0,toolEtna\WObj:=wobjEtna;
    TriggL T1203,vl,laserOFF,z0,toolEtna\WObj:=wobjEtna;
    TriggL T1204,v50,laserON,z0,toolEtna\WObj:=wobjEtna;
    TriggL T1205,vl,laserOFF,z0,toolEtna\WObj:=wobjEtna;
    TriggL T1206,v50,laserON,z0,toolEtna\WObj:=wobjEtna;
    TriggL T1207,vl,laserOFF,z0,toolEtna\WObj:=wobjEtna;
    TriggL T1208,v50,laserON,z0,toolEtna\WObj:=wobjEtna;
    TriggL T1209,vl,laserOFF,z0,toolEtna\WObj:=wobjEtna;
    TriggL T1210,v50,laserON,z0,toolEtna\WObj:=wobjEtna;
    TriggL T1211,vl,laserOFF,z0,toolEtna\WObj:=wobjEtna;
    TriggL T1212,v50,laserON,z0,toolEtna\WObj:=wobjEtna;
    TriggL T1213,vl,laserOFF,z0,toolEtna\WObj:=wobjEtna;
    TriggL T1214,v50,laserON,z0,toolEtna\WObj:=wobjEtna;
    TriggL T1215,vl,laserOFF,z0,toolEtna\WObj:=wobjEtna;
    TriggL T1216,v50,laserON,z0,toolEtna\WObj:=wobjEtna;
    TriggL T1217,vl,laserOFF,z0,toolEtna\WObj:=wobjEtna;
    TriggL T1218,v50,laserON,z0,toolEtna\WObj:=wobjEtna;
    TriggL T1219,vl,laserOFF,z0,toolEtna\WObj:=wobjEtna;
    TriggL T1220,v50,laserON,z0,toolEtna\WObj:=wobjEtna;
    TriggL T1221,vl,laserOFF,z0,toolEtna\WObj:=wobjEtna;
    TriggL T1222,v50,laserON,z0,toolEtna\WObj:=wobjEtna;
    TriggL T1223,vl,laserOFF,z0,toolEtna\WObj:=wobjEtna;
    TriggL T1224,v50,laserON,z0,toolEtna\WObj:=wobjEtna;
    TriggL T1225,vl,laserOFF,z0,toolEtna\WObj:=wobjEtna;
    TriggL T1226,v50,laserON,z0,toolEtna\WObj:=wobjEtna;
    TriggL T1227,vl,laserOFF,z0,toolEtna\WObj:=wobjEtna;
    TriggL T1228,v50,laserON,z0,toolEtna\WObj:=wobjEtna;
    TriggL T1229,vl,laserOFF,z0,toolEtna\WObj:=wobjEtna;
    TriggL T1230,v50,laserON,z0,toolEtna\WObj:=wobjEtna;
    TriggL T1231,vl,laserOFF,z0,toolEtna\WObj:=wobjEtna;
    TriggL T1232,v50,laserON,z0,toolEtna\WObj:=wobjEtna;
    TriggL T1233,vl,laserOFF,z0,toolEtna\WObj:=wobjEtna;
    TriggL T1234,v50,laserON,z0,toolEtna\WObj:=wobjEtna;
    TriggL T1235,vl,laserOFF,z0,toolEtna\WObj:=wobjEtna;
    TriggL T1236,v50,laserON,z0,toolEtna\WObj:=wobjEtna;
    TriggL T1237,vl,laserOFF,z0,toolEtna\WObj:=wobjEtna;
    TriggL T1238,v50,laserON,z0,toolEtna\WObj:=wobjEtna;
    TriggL T1239,vl,laserOFF,z0,toolEtna\WObj:=wobjEtna;
    TriggL T1240,v50,laserON,z0,toolEtna\WObj:=wobjEtna;
    TriggL T1241,vl,laserOFF,z0,toolEtna\WObj:=wobjEtna;
    TriggL T1242,v50,laserON,z0,toolEtna\WObj:=wobjEtna;
    TriggL T1243,vl,laserOFF,z0,toolEtna\WObj:=wobjEtna;
    TriggL T1244,v50,laserON,z0,toolEtna\WObj:=wobjEtna;
    TriggL T1245,vl,laserOFF,z0,toolEtna\WObj:=wobjEtna;
    TriggL T1246,v50,laserON,z0,toolEtna\WObj:=wobjEtna;
    TriggL T1247,vl,laserOFF,z0,toolEtna\WObj:=wobjEtna;
    TriggL T1248,v50,laserON,z0,toolEtna\WObj:=wobjEtna;
    TriggL T1249,vl,laserOFF,z0,toolEtna\WObj:=wobjEtna;
    TriggL T1250,v50,laserON,z0,toolEtna\WObj:=wobjEtna;
    TriggL T1251,vl,laserOFF,z0,toolEtna\WObj:=wobjEtna;
    TriggL T1252,v50,laserON,z0,toolEtna\WObj:=wobjEtna;
    TriggL T1253,vl,laserOFF,z0,toolEtna\WObj:=wobjEtna;
    TriggL T1254,v50,laserON,z0,toolEtna\WObj:=wobjEtna;
    TriggL T1255,vl,laserOFF,z0,toolEtna\WObj:=wobjEtna;
    TriggL T1256,v50,laserON,z0,toolEtna\WObj:=wobjEtna;
    TriggL T1257,vl,laserOFF,z0,toolEtna\WObj:=wobjEtna;
    TriggL T1258,v50,laserON,z0,toolEtna\WObj:=wobjEtna;
    TriggL T1259,vl,laserOFF,z0,toolEtna\WObj:=wobjEtna;
    TriggL T1260,v50,laserON,z0,toolEtna\WObj:=wobjEtna;
    TriggL T1261,vl,laserOFF,z0,toolEtna\WObj:=wobjEtna;
    TriggL T1262,v50,laserON,z0,toolEtna\WObj:=wobjEtna;
    TriggL T1263,vl,laserOFF,z0,toolEtna\WObj:=wobjEtna;
    TriggL T1264,v50,laserON,z0,toolEtna\WObj:=wobjEtna;
    TriggL T1265,vl,laserOFF,z0,toolEtna\WObj:=wobjEtna;
    TriggL T1266,v50,laserON,z0,toolEtna\WObj:=wobjEtna;
    TriggL T1267,vl,laserOFF,z0,toolEtna\WObj:=wobjEtna;
    TriggL T1268,v50,laserON,z0,toolEtna\WObj:=wobjEtna;
    TriggL T1269,vl,laserOFF,z0,toolEtna\WObj:=wobjEtna;
    TriggL T1270,v50,laserON,z0,toolEtna\WObj:=wobjEtna;
    TriggL T1271,vl,laserOFF,z0,toolEtna\WObj:=wobjEtna;
    TriggL T1272,v50,laserON,z0,toolEtna\WObj:=wobjEtna;
    TriggL T1273,vl,laserOFF,z0,toolEtna\WObj:=wobjEtna;
    TriggL T1274,v50,laserON,z0,toolEtna\WObj:=wobjEtna;
    TriggL T1275,vl,laserOFF,z0,toolEtna\WObj:=wobjEtna;
    TriggL T1276,v50,laserON,z0,toolEtna\WObj:=wobjEtna;
    TriggL T1277,vl,laserOFF,z0,toolEtna\WObj:=wobjEtna;
    TriggL T1278,v50,laserON,z0,toolEtna\WObj:=wobjEtna;
    TriggL T1279,vl,laserOFF,z0,toolEtna\WObj:=wobjEtna;
    TriggL T1280,v50,laserON,z0,toolEtna\WObj:=wobjEtna;
    TriggL T1281,vl,laserOFF,z0,toolEtna\WObj:=wobjEtna;
    TriggL T1282,v50,laserON,z0,toolEtna\WObj:=wobjEtna;
    TriggL T1283,vl,laserOFF,z0,toolEtna\WObj:=wobjEtna;
    TriggL T1284,v50,laserON,z0,toolEtna\WObj:=wobjEtna;
    TriggL T1285,vl,laserOFF,z0,toolEtna\WObj:=wobjEtna;
    TriggL T1286,v50,laserON,z0,toolEtna\WObj:=wobjEtna;
    TriggL T1287,vl,laserOFF,z0,toolEtna\WObj:=wobjEtna;
    TriggL T1288,v50,laserON,z0,toolEtna\WObj:=wobjEtna;
    TriggL T1289,vl,laserOFF,z0,toolEtna\WObj:=wobjEtna;
    TriggL T1290,v50,laserON,z0,toolEtna\WObj:=wobjEtna;
    TriggL T1291,vl,laserOFF,z0,toolEtna\WObj:=wobjEtna;
    TriggL T1292,v50,laserON,z0,toolEtna\WObj:=wobjEtna;
    TriggL T1293,vl,laserOFF,z0,toolEtna\WObj:=wobjEtna;
    TriggL T1294,v50,laserON,z0,toolEtna\WObj:=wobjEtna;
    TriggL T1295,vl,laserOFF,z0,toolEtna\WObj:=wobjEtna;
    TriggL T1296,v50,laserON,z0,toolEtna\WObj:=wobjEtna;
    TriggL T1297,vl,laserOFF,z0,toolEtna\WObj:=wobjEtna;
    TriggL T1298,v50,laserON,z0,toolEtna\WObj:=wobjEtna;
    TriggL T1299,vl,laserOFF,z0,toolEtna\WObj:=wobjEtna;
    TriggL T1300,v50,laserON,z0,toolEtna\WObj:=wobjEtna;
    TriggL T1301,vl,laserOFF,z0,toolEtna\WObj:=wobjEtna;
    TriggL T1302,v50,laserON,z0,toolEtna\WObj:=wobjEtna;
    TriggL T1303,vl,laserOFF,z0,toolEtna\WObj:=wobjEtna;
    TriggL T1304,v50,laserON,z0,toolEtna\WObj:=wobjEtna;
    TriggL T1305,vl,laserOFF,z0,toolEtna\WObj:=wobjEtna;
    TriggL T1306,v50,laserON,z0,toolEtna\WObj:=wobjEtna;
    TriggL T1307,vl,laserOFF,z0,toolEtna\WObj:=wobjEtna;
    TriggL T1308,v50,laserON,z0,toolEtna\WObj:=wobjEtna;
    TriggL T1309,vl,laserOFF,z0,toolEtna\WObj:=wobjEtna;
    TriggL T1310,v50,laserON,z0,toolEtna\WObj:=wobjEtna;
    TriggL T1311,vl,laserOFF,z0,toolEtna\WObj:=wobjEtna;
    TriggL T1312,v50,laserON,z0,toolEtna\WObj:=wobjEtna;
    TriggL T1313,vl,laserOFF,z0,toolEtna\WObj:=wobjEtna;
    TriggL T1314,v50,laserON,z0,toolEtna\WObj:=wobjEtna;
    TriggL T1315,vl,laserOFF,z0,toolEtna\WObj:=wobjEtna;
    TriggL T1316,v50,laserON,z0,toolEtna\WObj:=wobjEtna;
    TriggL T1317,vl,laserOFF,z0,toolEtna\WObj:=wobjEtna;
    TriggL T1318,v50,laserON,z0,toolEtna\WObj:=wobjEtna;
    TriggL T1319,vl,laserOFF,z0,toolEtna\WObj:=wobjEtna;
    TriggL T1320,v50,laserON,z0,toolEtna\WObj:=wobjEtna;
    TriggL T1321,vl,laserOFF,z0,toolEtna\WObj:=wobjEtna;
    TriggL T1322,v50,laserON,z0,toolEtna\WObj:=wobjEtna;
    TriggL T1323,vl,laserOFF,z0,toolEtna\WObj:=wobjEtna;
    TriggL T1324,v50,laserON,z0,toolEtna\WObj:=wobjEtna;
    TriggL T1325,vl,laserOFF,z0,toolEtna\WObj:=wobjEtna;
    TriggL T1326,v50,laserON,z0,toolEtna\WObj:=wobjEtna;
    TriggL T1327,vl,laserOFF,z0,toolEtna\WObj:=wobjEtna;
    TriggL T1328,v50,laserON,z0,toolEtna\WObj:=wobjEtna;
    TriggL T1329,vl,laserOFF,z0,toolEtna\WObj:=wobjEtna;
    TriggL T1330,v50,laserON,z0,toolEtna\WObj:=wobjEtna;
    TriggL T1331,vl,laserOFF,z0,toolEtna\WObj:=wobjEtna;
    TriggL T1332,v50,laserON,z0,toolEtna\WObj:=wobjEtna;
    TriggL T1333,vl,laserOFF,z0,toolEtna\WObj:=wobjEtna;
    TriggL T1334,v50,laserON,z0,toolEtna\WObj:=wobjEtna;
    TriggL T1335,vl,laserOFF,z0,toolEtna\WObj:=wobjEtna;
    TriggL T1336,v50,laserON,z0,toolEtna\WObj:=wobjEtna;
    TriggL T1337,vl,laserOFF,z0,toolEtna\WObj:=wobjEtna;
    TriggL T1338,v50,laserON,z0,toolEtna\WObj:=wobjEtna;
    TriggL T1339,vl,laserOFF,z0,toolEtna\WObj:=wobjEtna;
    TriggL T1340,v50,laserON,z0,toolEtna\WObj:=wobjEtna;
    TriggL T1341,vl,laserOFF,z0,toolEtna\WObj:=wobjEtna;
    TriggL T1342,v50,laserON,z0,toolEtna\WObj:=wobjEtna;
    TriggL T1343,vl,laserOFF,z0,toolEtna\WObj:=wobjEtna;
    TriggL T1344,v50,laserON,z0,toolEtna\WObj:=wobjEtna;
    TriggL T1345,vl,laserOFF,z0,toolEtna\WObj:=wobjEtna;
    TriggL T1346,v50,laserON,z0,toolEtna\WObj:=wobjEtna;
    TriggL T1347,vl,laserOFF,z0,toolEtna\WObj:=wobjEtna;
    TriggL T1348,v50,laserON,z0,toolEtna\WObj:=wobjEtna;
    TriggL T1349,vl,laserOFF,z0,toolEtna\WObj:=wobjEtna;
    TriggL T1350,v50,laserON,z0,toolEtna\WObj:=wobjEtna;
    TriggL T1351,vl,laserOFF,z0,toolEtna\WObj:=wobjEtna;
    TriggL T1352,v50,laserON,z0,toolEtna\WObj:=wobjEtna;
    TriggL T1353,vl,laserOFF,z0,toolEtna\WObj:=wobjEtna;
    TriggL T1354,v50,laserON,z0,toolEtna\WObj:=wobjEtna;
    TriggL T1355,vl,laserOFF,z0,toolEtna\WObj:=wobjEtna;
    TriggL T1356,v50,laserON,z0,toolEtna\WObj:=wobjEtna;
    TriggL T1357,vl,laserOFF,z0,toolEtna\WObj:=wobjEtna;
    TriggL T1358,v50,laserON,z0,toolEtna\WObj:=wobjEtna;
    TriggL T1359,vl,laserOFF,z0,toolEtna\WObj:=wobjEtna;
    TriggL T1360,v50,laserON,z0,toolEtna\WObj:=wobjEtna;
    TriggL T1361,vl,laserOFF,z0,toolEtna\WObj:=wobjEtna;
    TriggL T1362,v50,laserON,z0,toolEtna\WObj:=wobjEtna;
    TriggL T1363,vl,laserOFF,z0,toolEtna\WObj:=wobjEtna;
    TriggL T1364,v50,laserON,z0,toolEtna\WObj:=wobjEtna;
    TriggL T1365,vl,laserOFF,z0,toolEtna\WObj:=wobjEtna;
    TriggL T1366,v50,laserON,z0,toolEtna\WObj:=wobjEtna;
    TriggL T1367,vl,laserOFF,z0,toolEtna\WObj:=wobjEtna;
    TriggL T1368,v50,laserON,z0,toolEtna\WObj:=wobjEtna;
    TriggL T1369,vl,laserOFF,z0,toolEtna\WObj:=wobjEtna;
    TriggL T1370,v50,laserON,z0,toolEtna\WObj:=wobjEtna;
    TriggL T1371,vl,laserOFF,z0,toolEtna\WObj:=wobjEtna;
    TriggL T1372,v50,laserON,z0,toolEtna\WObj:=wobjEtna;
    TriggL T1373,vl,laserOFF,z0,toolEtna\WObj:=wobjEtna;
    TriggL T1374,v50,laserON,z0,toolEtna\WObj:=wobjEtna;
    TriggL T1375,vl,laserOFF,z0,toolEtna\WObj:=wobjEtna;
    TriggL T1376,v50,laserON,z0,toolEtna\WObj:=wobjEtna;
    TriggL T1377,vl,laserOFF,z0,toolEtna\WObj:=wobjEtna;
    TriggL T1378,v50,laserON,z0,toolEtna\WObj:=wobjEtna;
    TriggL T1379,vl,laserOFF,z0,toolEtna\WObj:=wobjEtna;
    TriggL T1380,v50,laserON,z0,toolEtna\WObj:=wobjEtna;
    TriggL T1381,vl,laserOFF,z0,toolEtna\WObj:=wobjEtna;
    TriggL T1382,v50,laserON,z0,toolEtna\WObj:=wobjEtna;
    TriggL T1383,vl,laserOFF,z0,toolEtna\WObj:=wobjEtna;
    TriggL T1384,v50,laserON,z0,toolEtna\WObj:=wobjEtna;
    TriggL T1385,vl,laserOFF,z0,toolEtna\WObj:=wobjEtna;
    TriggL T1386,v50,laserON,z0,toolEtna\WObj:=wobjEtna;
    TriggL T1387,vl,laserOFF,z0,toolEtna\WObj:=wobjEtna;
    TriggL T1388,v50,laserON,z0,toolEtna\WObj:=wobjEtna;
    TriggL T1389,vl,laserOFF,z0,toolEtna\WObj:=wobjEtna;
    TriggL T1390,v50,laserON,z0,toolEtna\WObj:=wobjEtna;
    TriggL T1391,vl,laserOFF,z0,toolEtna\WObj:=wobjEtna;
    TriggL T1392,v50,laserON,z0,toolEtna\WObj:=wobjEtna;
    TriggL T1393,vl,laserOFF,z0,toolEtna\WObj:=wobjEtna;
    TriggL T1394,v50,laserON,z0,toolEtna\WObj:=wobjEtna;
    TriggL T1395,vl,laserOFF,z0,toolEtna\WObj:=wobjEtna;
    TriggL T1396,v50,laserON,z0,toolEtna\WObj:=wobjEtna;
    TriggL T1397,vl,laserOFF,z0,toolEtna\WObj:=wobjEtna;
    TriggL T1398,v50,laserON,z0,toolEtna\WObj:=wobjEtna;
    TriggL T1399,vl,laserOFF,z0,toolEtna\WObj:=wobjEtna;
    TriggL T1400,v50,laserON,z0,toolEtna\WObj:=wobjEtna;
    TriggL T1401,vl,laserOFF,z0,toolEtna\WObj:=wobjEtna;
    TriggL T1402,v50,laserON,z0,toolEtna\WObj:=wobjEtna;
    TriggL T1403,vl,laserOFF,z0,toolEtna\WObj:=wobjEtna;
    TriggL T1404,v50,laserON,z0,toolEtna\WObj:=wobjEtna;
    TriggL T1405,vl,laserOFF,z0,toolEtna\WObj:=wobjEtna;
    TriggL T1406,v50,laserON,z0,toolEtna\WObj:=wobjEtna;
    TriggL T1407,vl,laserOFF,z0,toolEtna\WObj:=wobjEtna;
    TriggL T1408,v50,laserON,z0,toolEtna\WObj:=wobjEtna;
    TriggL T1409,vl,laserOFF,z0,toolEtna\WObj:=wobjEtna;
    TriggL T1410,v50,laserON,z0,toolEtna\WObj:=wobjEtna;
    TriggL T1411,vl,laserOFF,z0,toolEtna\WObj:=wobjEtna;
    TriggL T1412,v50,laserON,z0,toolEtna\WObj:=wobjEtna;
    TriggL T1413,vl,laserOFF,z0,toolEtna\WObj:=wobjEtna;
    TriggL T1414,v50,laserON,z0,toolEtna\WObj:=wobjEtna;
    TriggL T1415,vl,laserOFF,z0,toolEtna\WObj:=wobjEtna;
    TriggL T1416,v50,laserON,z0,toolEtna\WObj:=wobjEtna;
    TriggL T1417,vl,laserOFF,z0,toolEtna\WObj:=wobjEtna;
    TriggL T1418,v50,laserON,z0,toolEtna\WObj:=wobjEtna;
    TriggL T1419,vl,laserOFF,z0,toolEtna\WObj:=wobjEtna;
    TriggL T1420,v50,laserON,z0,toolEtna\WObj:=wobjEtna;
    TriggL T1421,vl,laserOFF,z0,toolEtna\WObj:=wobjEtna;
    TriggL T1422,v50,laserON,z0,toolEtna\WObj:=wobjEtna;
    TriggL T1423,vl,laserOFF,z0,toolEtna\WObj:=wobjEtna;
    TriggL T1424,v50,laserON,z0,toolEtna\WObj:=wobjEtna;
    TriggL T1425,vl,laserOFF,z0,toolEtna\WObj:=wobjEtna;
    TriggL T1426,v50,laserON,z0,toolEtna\WObj:=wobjEtna;
    TriggL T1427,vl,laserOFF,z0,toolEtna\WObj:=wobjEtna;
    TriggL T1428,v50,laserON,z0,toolEtna\WObj:=wobjEtna;
    TriggL T1429,vl,laserOFF,z0,toolEtna\WObj:=wobjEtna;
    TriggL T1430,v50,laserON,z0,toolEtna\WObj:=wobjEtna;
    TriggL T1431,vl,laserOFF,z0,toolEtna\WObj:=wobjEtna;
    TriggL T1432,v50,laserON,z0,toolEtna\WObj:=wobjEtna;
    TriggL T1433,vl,laserOFF,z0,toolEtna\WObj:=wobjEtna;
    TriggL T1434,v50,laserON,z0,toolEtna\WObj:=wobjEtna;
    TriggL T1435,vl,laserOFF,z0,toolEtna\WObj:=wobjEtna;
    TriggL T1436,v50,laserON,z0,toolEtna\WObj:=wobjEtna;
    TriggL T1437,vl,laserOFF,z0,toolEtna\WObj:=wobjEtna;
    TriggL T1438,v50,laserON,z0,toolEtna\WObj:=wobjEtna;
    TriggL T1439,vl,laserOFF,z0,toolEtna\WObj:=wobjEtna;
    TriggL T1440,v50,laserON,z0,toolEtna\WObj:=wobjEtna;
    TriggL T1441,vl,laserOFF,z0,toolEtna\WObj:=wobjEtna;
    TriggL T1442,v50,laserON,z0,toolEtna\WObj:=wobjEtna;
    TriggL T1443,vl,laserOFF,z0,toolEtna\WObj:=wobjEtna;
    TriggL T1444,v50,laserON,z0,toolEtna\WObj:=wobjEtna;
    TriggL T1445,vl,laserOFF,z0,toolEtna\WObj:=wobjEtna;
    TriggL T1446,v50,laserON,z0,toolEtna\WObj:=wobjEtna;
    TriggL T1447,vl,laserOFF,z0,toolEtna\WObj:=wobjEtna;
    TriggL T1448,v50,laserON,z0,toolEtna\WObj:=wobjEtna;
    TriggL T1449,vl,laserOFF,z0,toolEtna\WObj:=wobjEtna;
    TriggL T1450,v50,laserON,z0,toolEtna\WObj:=wobjEtna;
    TriggL T1451,vl,laserOFF,z0,toolEtna\WObj:=wobjEtna;
    TriggL T1452,v50,laserON,z0,toolEtna\WObj:=wobjEtna;
    TriggL T1453,vl,laserOFF,z0,toolEtna\WObj:=wobjEtna;
    TriggL T1454,v50,laserON,z0,toolEtna\WObj:=wobjEtna;
    TriggL T1455,vl,laserOFF,z0,toolEtna\WObj:=wobjEtna;
    TriggL T1456,v50,laserON,z0,toolEtna\WObj:=wobjEtna;
    TriggL T1457,vl,laserOFF,z0,toolEtna\WObj:=wobjEtna;
    TriggL T1458,v50,laserON,z0,toolEtna\WObj:=wobjEtna;
    TriggL T1459,vl,laserOFF,z0,toolEtna\WObj:=wobjEtna;
    TriggL T1460,v50,laserON,z0,toolEtna\WObj:=wobjEtna;
    TriggL T1461,vl,laserOFF,z0,toolEtna\WObj:=wobjEtna;
    TriggL T1462,v50,laserON,z0,toolEtna\WObj:=wobjEtna;
    TriggL T1463,vl,laserOFF,z0,toolEtna\WObj:=wobjEtna;
    TriggL T1464,v50,laserON,z0,toolEtna\WObj:=wobjEtna;
    TriggL T1465,vl,laserOFF,z0,toolEtna\WObj:=wobjEtna;
    TriggL T1466,v50,laserON,z0,toolEtna\WObj:=wobjEtna;
    TriggL T1467,vl,laserOFF,z0,toolEtna\WObj:=wobjEtna;
    TriggL T1468,v50,laserON,z0,toolEtna\WObj:=wobjEtna;
    TriggL T1469,vl,laserOFF,z0,toolEtna\WObj:=wobjEtna;
    TriggL T1470,v50,laserON,z0,toolEtna\WObj:=wobjEtna;
    TriggL T1471,vl,laserOFF,z0,toolEtna\WObj:=wobjEtna;
    TriggL T1472,v50,laserON,z0,toolEtna\WObj:=wobjEtna;
    TriggL T1473,vl,laserOFF,z0,toolEtna\WObj:=wobjEtna;
    TriggL T1474,v50,laserON,z0,toolEtna\WObj:=wobjEtna;
    TriggL T1475,vl,laserOFF,z0,toolEtna\WObj:=wobjEtna;
    TriggL T1476,v50,laserON,z0,toolEtna\WObj:=wobjEtna;
    TriggL T1477,vl,laserOFF,z0,toolEtna\WObj:=wobjEtna;
    TriggL T1478,v50,laserON,z0,toolEtna\WObj:=wobjEtna;
    TriggL T1479,vl,laserOFF,z0,toolEtna\WObj:=wobjEtna;
    TriggL T1480,v50,laserON,z0,toolEtna\WObj:=wobjEtna;
    TriggL T1481,vl,laserOFF,z0,toolEtna\WObj:=wobjEtna;
    TriggL T1482,v50,laserON,z0,toolEtna\WObj:=wobjEtna;
    TriggL T1483,vl,laserOFF,z0,toolEtna\WObj:=wobjEtna;
    TriggL T1484,v50,laserON,z0,toolEtna\WObj:=wobjEtna;
    TriggL T1485,vl,laserOFF,z0,toolEtna\WObj:=wobjEtna;
    TriggL T1486,v50,laserON,z0,toolEtna\WObj:=wobjEtna;
    TriggL T1487,vl,laserOFF,z0,toolEtna\WObj:=wobjEtna;
    TriggL T1488,v50,laserON,z0,toolEtna\WObj:=wobjEtna;
    TriggL T1489,vl,laserOFF,z0,toolEtna\WObj:=wobjEtna;
    TriggL T1490,v50,laserON,z0,toolEtna\WObj:=wobjEtna;
    TriggL T1491,vl,laserOFF,z0,toolEtna\WObj:=wobjEtna;
    TriggL T1492,v50,laserON,z0,toolEtna\WObj:=wobjEtna;
    TriggL T1493,vl,laserOFF,z0,toolEtna\WObj:=wobjEtna;
    TriggL T1494,v50,laserON,z0,toolEtna\WObj:=wobjEtna;
    TriggL T1495,vl,laserOFF,z0,toolEtna\WObj:=wobjEtna;
    TriggL T1496,v50,laserON,z0,toolEtna\WObj:=wobjEtna;
    TriggL T1497,vl,laserOFF,z0,toolEtna\WObj:=wobjEtna;
    TriggL T1498,v50,laserON,z0,toolEtna\WObj:=wobjEtna;
    TriggL T1499,vl,laserOFF,z0,toolEtna\WObj:=wobjEtna;
    TriggL T1500,v50,laserON,z0,toolEtna\WObj:=wobjEtna;
    TriggL T1501,vl,laserOFF,z0,toolEtna\WObj:=wobjEtna;
    TriggL T1502,v50,laserON,z0,toolEtna\WObj:=wobjEtna;
    TriggL T1503,vl,laserOFF,z0,toolEtna\WObj:=wobjEtna;
    TriggL T1504,v50,laserON,z0,toolEtna\WObj:=wobjEtna;
    TriggL T1505,vl,laserOFF,z0,toolEtna\WObj:=wobjEtna;
    TriggL T1506,v50,laserON,z0,toolEtna\WObj:=wobjEtna;
    TriggL T1507,vl,laserOFF,z0,toolEtna\WObj:=wobjEtna;
    TriggL T1508,v50,laserON,z0,toolEtna\WObj:=wobjEtna;
    TriggL T1509,vl,laserOFF,z0,toolEtna\WObj:=wobjEtna;
    TriggL T1510,v50,laserON,z0,toolEtna\WObj:=wobjEtna;
    TriggL T1511,vl,laserOFF,z0,toolEtna\WObj:=wobjEtna;
    TriggL T1512,v50,laserON,z0,toolEtna\WObj:=wobjEtna;
    TriggL T1513,vl,laserOFF,z0,toolEtna\WObj:=wobjEtna;
    TriggL T1514,v50,laserON,z0,toolEtna\WObj:=wobjEtna;
    TriggL T1515,vl,laserOFF,z0,toolEtna\WObj:=wobjEtna;
    TriggL T1516,v50,laserON,z0,toolEtna\WObj:=wobjEtna;
    TriggL T1517,vl,laserOFF,z0,toolEtna\WObj:=wobjEtna;
    TriggL T1518,v50,laserON,z0,toolEtna\WObj:=wobjEtna;
    TriggL T1519,vl,laserOFF,z0,toolEtna\WObj:=wobjEtna;
    TriggL T1520,v50,laserON,z0,toolEtna\WObj:=wobjEtna;
    TriggL T1521,vl,laserOFF,z0,toolEtna\WObj:=wobjEtna;
    TriggL T1522,v50,laserON,z0,toolEtna\WObj:=wobjEtna;
    TriggL T1523,vl,laserOFF,z0,toolEtna\WObj:=wobjEtna;
    TriggL T1524,v50,laserON,z0,toolEtna\WObj:=wobjEtna;
    TriggL T1525,vl,laserOFF,z0,toolEtna\WObj:=wobjEtna;
    TriggL T1526,v50,laserON,z0,toolEtna\WObj:=wobjEtna;
    TriggL T1527,vl,laserOFF,z0,toolEtna\WObj:=wobjEtna;
    TriggL T1528,v50,laserON,z0,toolEtna\WObj:=wobjEtna;
    TriggL T1529,vl,laserOFF,z0,toolEtna\WObj:=wobjEtna;
    TriggL T1530,v50,laserON,z0,toolEtna\WObj:=wobjEtna;
    TriggL T1531,vl,laserOFF,z0,toolEtna\WObj:=wobjEtna;
    TriggL T1532,v50,laserON,z0,toolEtna\WObj:=wobjEtna;
    TriggL T1533,vl,laserOFF,z0,toolEtna\WObj:=wobjEtna;
    TriggL T1534,v50,laserON,z0,toolEtna\WObj:=wobjEtna;
    TriggL T1535,vl,laserOFF,z0,toolEtna\WObj:=wobjEtna;
    TriggL T1536,v50,laserON,z0,toolEtna\WObj:=wobjEtna;
    TriggL T1537,vl,laserOFF,z0,toolEtna\WObj:=wobjEtna;
    TriggL T1538,v50,laserON,z0,toolEtna\WObj:=wobjEtna;
    TriggL T1539,vl,laserOFF,z0,toolEtna\WObj:=wobjEtna;
    TriggL T1540,v50,laserON,z0,toolEtna\WObj:=wobjEtna;
    TriggL T1541,vl,laserOFF,z0,toolEtna\WObj:=wobjEtna;
    TriggL T1542,v50,laserON,z0,toolEtna\WObj:=wobjEtna;
    TriggL T1543,vl,laserOFF,z0,toolEtna\WObj:=wobjEtna;
    TriggL T1544,v50,laserON,z0,toolEtna\WObj:=wobjEtna;
    TriggL T1545,vl,laserOFF,z0,toolEtna\WObj:=wobjEtna;
    TriggL T1546,v50,laserON,z0,toolEtna\WObj:=wobjEtna;
    TriggL T1547,vl,laserOFF,z0,toolEtna\WObj:=wobjEtna;
    TriggL T1548,v50,laserON,z0,toolEtna\WObj:=wobjEtna;
    TriggL T1549,vl,laserOFF,z0,toolEtna\WObj:=wobjEtna;
    TriggL T1550,v50,laserON,z0,toolEtna\WObj:=wobjEtna;
    TriggL T1551,vl,laserOFF,z0,toolEtna\WObj:=wobjEtna;
    TriggL T1552,v50,laserON,z0,toolEtna\WObj:=wobjEtna;
    TriggL T1553,vl,laserOFF,z0,toolEtna\WObj:=wobjEtna;
    TriggL T1554,v50,laserON,z0,toolEtna\WObj:=wobjEtna;
    TriggL T1555,vl,laserOFF,z0,toolEtna\WObj:=wobjEtna;
    TriggL T1556,v50,laserON,z0,toolEtna\WObj:=wobjEtna;
    TriggL T1557,vl,laserOFF,z0,toolEtna\WObj:=wobjEtna;
    TriggL T1558,v50,laserON,z0,toolEtna\WObj:=wobjEtna;
    TriggL T1559,vl,laserOFF,z0,toolEtna\WObj:=wobjEtna;
    TriggL T1560,v50,laserON,z0,toolEtna\WObj:=wobjEtna;
    TriggL T1561,vl,laserOFF,z0,toolEtna\WObj:=wobjEtna;
    TriggL T1562,v50,laserON,z0,toolEtna\WObj:=wobjEtna;
    TriggL T1563,vl,laserOFF,z0,toolEtna\WObj:=wobjEtna;
    TriggL T1564,v50,laserON,z0,toolEtna\WObj:=wobjEtna;
    TriggL T1565,vl,laserOFF,z0,toolEtna\WObj:=wobjEtna;
    TriggL T1566,v50,laserON,z0,toolEtna\WObj:=wobjEtna;
    TriggL T1567,vl,laserOFF,z0,toolEtna\WObj:=wobjEtna;
    TriggL T1568,v50,laserON,z0,toolEtna\WObj:=wobjEtna;
    TriggL T1569,vl,laserOFF,z0,toolEtna\WObj:=wobjEtna;
    TriggL T1570,v50,laserON,z0,toolEtna\WObj:=wobjEtna;
    TriggL T1571,vl,laserOFF,z0,toolEtna\WObj:=wobjEtna;
    TriggL T1572,v50,laserON,z0,toolEtna\WObj:=wobjEtna;
    TriggL T1573,vl,laserOFF,z0,toolEtna\WObj:=wobjEtna;
    TriggL T1574,v50,laserON,z0,toolEtna\WObj:=wobjEtna;
    TriggL T1575,vl,laserOFF,z0,toolEtna\WObj:=wobjEtna;
    TriggL T1576,v50,laserON,z0,toolEtna\WObj:=wobjEtna;
    TriggL T1577,vl,laserOFF,z0,toolEtna\WObj:=wobjEtna;
    TriggL T1578,v50,laserON,z0,toolEtna\WObj:=wobjEtna;
    TriggL T1579,vl,laserOFF,z0,toolEtna\WObj:=wobjEtna;
    TriggL T1580,v50,laserON,z0,toolEtna\WObj:=wobjEtna;
    TriggL T1581,vl,laserOFF,z0,toolEtna\WObj:=wobjEtna;
    TriggL T1582,v50,laserON,z0,toolEtna\WObj:=wobjEtna;
    TriggL T1583,vl,laserOFF,z0,toolEtna\WObj:=wobjEtna;
    TriggL T1584,v50,laserON,z0,toolEtna\WObj:=wobjEtna;
    TriggL T1585,vl,laserOFF,z0,toolEtna\WObj:=wobjEtna;
    TriggL T1586,v50,laserON,z0,toolEtna\WObj:=wobjEtna;
    TriggL T1587,vl,laserOFF,z0,toolEtna\WObj:=wobjEtna;
    TriggL T1588,v50,laserON,z0,toolEtna\WObj:=wobjEtna;
    TriggL T1589,vl,laserOFF,z0,toolEtna\WObj:=wobjEtna;
    TriggL T1590,v50,laserON,z0,toolEtna\WObj:=wobjEtna;
    TriggL T1591,vl,laserOFF,z0,toolEtna\WObj:=wobjEtna;
    TriggL T1592,v50,laserON,z0,toolEtna\WObj:=wobjEtna;
    TriggL T1593,vl,laserOFF,z0,toolEtna\WObj:=wobjEtna;
    TriggL T1594,v50,laserON,z0,toolEtna\WObj:=wobjEtna;
    TriggL T1595,vl,laserOFF,z0,toolEtna\WObj:=wobjEtna;
    TriggL T1596,v50,laserON,z0,toolEtna\WObj:=wobjEtna;
    TriggL T1597,vl,laserOFF,z0,toolEtna\WObj:=wobjEtna;
    TriggL T1598,v50,laserON,z0,toolEtna\WObj:=wobjEtna;
    TriggL T1599,vl,laserOFF,z0,toolEtna\WObj:=wobjEtna;
    TriggL T1600,v50,laserON,z0,toolEtna\WObj:=wobjEtna;
    TriggL T1601,vl,laserOFF,z0,toolEtna\WObj:=wobjEtna;
    TriggL T1602,v50,laserON,z0,toolEtna\WObj:=wobjEtna;
    TriggL T1603,vl,laserOFF,z0,toolEtna\WObj:=wobjEtna;
    TriggL T1604,v50,laserON,z0,toolEtna\WObj:=wobjEtna;
    TriggL T1605,vl,laserOFF,z0,toolEtna\WObj:=wobjEtna;
    TriggL T1606,v50,laserON,z0,toolEtna\WObj:=wobjEtna;
    TriggL T1607,vl,laserOFF,z0,toolEtna\WObj:=wobjEtna;
    TriggL T1608,v50,laserON,z0,toolEtna\WObj:=wobjEtna;
    TriggL T1609,vl,laserOFF,z0,toolEtna\WObj:=wobjEtna;
    TriggL T1610,v50,laserON,z0,toolEtna\WObj:=wobjEtna;
    TriggL T1611,vl,laserOFF,z0,toolEtna\WObj:=wobjEtna;
    TriggL T1612,v50,laserON,z0,toolEtna\WObj:=wobjEtna;
    TriggL T1613,vl,laserOFF,z0,toolEtna\WObj:=wobjEtna;
    TriggL T1614,v50,laserON,z0,toolEtna\WObj:=wobjEtna;
    TriggL T1615,vl,laserOFF,z0,toolEtna\WObj:=wobjEtna;
    TriggL T1616,v50,laserON,z0,toolEtna\WObj:=wobjEtna;
    TriggL T1617,vl,laserOFF,z0,toolEtna\WObj:=wobjEtna;
    TriggL T1618,v50,laserON,z0,toolEtna\WObj:=wobjEtna;
    TriggL T1619,vl,laserOFF,z0,toolEtna\WObj:=wobjEtna;
    TriggL T1620,v50,laserON,z0,toolEtna\WObj:=wobjEtna;
    TriggL T1621,vl,laserOFF,z0,toolEtna\WObj:=wobjEtna;
    TriggL T1622,v50,laserON,z0,toolEtna\WObj:=wobjEtna;
    TriggL T1623,vl,laserOFF,z0,toolEtna\WObj:=wobjEtna;
    TriggL T1624,v50,laserON,z0,toolEtna\WObj:=wobjEtna;
    TriggL T1625,vl,laserOFF,z0,toolEtna\WObj:=wobjEtna;
    TriggL T1626,v50,laserON,z0,toolEtna\WObj:=wobjEtna;
    TriggL T1627,vl,laserOFF,z0,toolEtna\WObj:=wobjEtna;
    TriggL T1628,v50,laserON,z0,toolEtna\WObj:=wobjEtna;
    TriggL T1629,vl,laserOFF,z0,toolEtna\WObj:=wobjEtna;
    TriggL T1630,v50,laserON,z0,toolEtna\WObj:=wobjEtna;
    TriggL T1631,vl,laserOFF,z0,toolEtna\WObj:=wobjEtna;
    TriggL T1632,v50,laserON,z0,toolEtna\WObj:=wobjEtna;
    TriggL T1633,vl,laserOFF,z0,toolEtna\WObj:=wobjEtna;
    TriggL T1634,v50,laserON,z0,toolEtna\WObj:=wobjEtna;
    TriggL T1635,vl,laserOFF,z0,toolEtna\WObj:=wobjEtna;
    TriggL T1636,v50,laserON,z0,toolEtna\WObj:=wobjEtna;
    TriggL T1637,vl,laserOFF,z0,toolEtna\WObj:=wobjEtna;
    TriggL T1638,v50,laserON,z0,toolEtna\WObj:=wobjEtna;
    TriggL T1639,vl,laserOFF,z0,toolEtna\WObj:=wobjEtna;
    TriggL T1640,v50,laserON,z0,toolEtna\WObj:=wobjEtna;
    TriggL T1641,vl,laserOFF,z0,toolEtna\WObj:=wobjEtna;
    TriggL T1642,v50,laserON,z0,toolEtna\WObj:=wobjEtna;
    TriggL T1643,vl,laserOFF,z0,toolEtna\WObj:=wobjEtna;
    TriggL T1644,v50,laserON,z0,toolEtna\WObj:=wobjEtna;
    TriggL T1645,vl,laserOFF,z0,toolEtna\WObj:=wobjEtna;
    TriggL T1646,v50,laserON,z0,toolEtna\WObj:=wobjEtna;
    TriggL T1647,vl,laserOFF,z0,toolEtna\WObj:=wobjEtna;
    TriggL T1648,v50,laserON,z0,toolEtna\WObj:=wobjEtna;
    TriggL T1649,vl,laserOFF,z0,toolEtna\WObj:=wobjEtna;
    TriggL T1650,v50,laserON,z0,toolEtna\WObj:=wobjEtna;
    TriggL T1651,vl,laserOFF,z0,toolEtna\WObj:=wobjEtna;
    TriggL T1652,v50,laserON,z0,toolEtna\WObj:=wobjEtna;
    TriggL T1653,vl,laserOFF,z0,toolEtna\WObj:=wobjEtna;
    TriggL T1654,v50,laserON,z0,toolEtna\WObj:=wobjEtna;
    TriggL T1655,vl,laserOFF,z0,toolEtna\WObj:=wobjEtna;
    TriggL T1656,v50,laserON,z0,toolEtna\WObj:=wobjEtna;
    TriggL T1657,vl,laserOFF,z0,toolEtna\WObj:=wobjEtna;
    TriggL T1658,v50,laserON,z0,toolEtna\WObj:=wobjEtna;
    TriggL T1659,vl,laserOFF,z0,toolEtna\WObj:=wobjEtna;
    TriggL T1660,v50,laserON,z0,toolEtna\WObj:=wobjEtna;
    TriggL T1661,vl,laserOFF,z0,toolEtna\WObj:=wobjEtna;
    TriggL T1662,v50,laserON,z0,toolEtna\WObj:=wobjEtna;
    TriggL T1663,vl,laserOFF,z0,toolEtna\WObj:=wobjEtna;
    TriggL T1664,v50,laserON,z0,toolEtna\WObj:=wobjEtna;
    TriggL T1665,vl,laserOFF,z0,toolEtna\WObj:=wobjEtna;
    TriggL T1666,v50,laserON,z0,toolEtna\WObj:=wobjEtna;
    TriggL T1667,vl,laserOFF,z0,toolEtna\WObj:=wobjEtna;
    TriggL T1668,v50,laserON,z0,toolEtna\WObj:=wobjEtna;
    TriggL T1669,vl,laserOFF,z0,toolEtna\WObj:=wobjEtna;
    TriggL T1670,v50,laserON,z0,toolEtna\WObj:=wobjEtna;
    TriggL T1671,vl,laserOFF,z0,toolEtna\WObj:=wobjEtna;
    TriggL T1672,v50,laserON,z0,toolEtna\WObj:=wobjEtna;
    TriggL T1673,vl,laserOFF,z0,toolEtna\WObj:=wobjEtna;
    TriggL T1674,v50,laserON,z0,toolEtna\WObj:=wobjEtna;
    TriggL T1675,vl,laserOFF,z0,toolEtna\WObj:=wobjEtna;
    TriggL T1676,v50,laserON,z0,toolEtna\WObj:=wobjEtna;
    TriggL T1677,vl,laserOFF,z0,toolEtna\WObj:=wobjEtna;
    TriggL T1678,v50,laserON,z0,toolEtna\WObj:=wobjEtna;
    TriggL T1679,vl,laserOFF,z0,toolEtna\WObj:=wobjEtna;
    TriggL T1680,v50,laserON,z0,toolEtna\WObj:=wobjEtna;
    TriggL T1681,vl,laserOFF,z0,toolEtna\WObj:=wobjEtna;
    TriggL T1682,v50,laserON,z0,toolEtna\WObj:=wobjEtna;
    TriggL T1683,vl,laserOFF,z0,toolEtna\WObj:=wobjEtna;
    TriggL T1684,v50,laserON,z0,toolEtna\WObj:=wobjEtna;
    TriggL T1685,vl,laserOFF,z0,toolEtna\WObj:=wobjEtna;
    TriggL T1686,v50,laserON,z0,toolEtna\WObj:=wobjEtna;
    TriggL T1687,vl,laserOFF,z0,toolEtna\WObj:=wobjEtna;
    TriggL T1688,v50,laserON,z0,toolEtna\WObj:=wobjEtna;
    TriggL T1689,vl,laserOFF,z0,toolEtna\WObj:=wobjEtna;
    TriggL T1690,v50,laserON,z0,toolEtna\WObj:=wobjEtna;
    TriggL T1691,vl,laserOFF,z0,toolEtna\WObj:=wobjEtna;
    TriggL T1692,v50,laserON,z0,toolEtna\WObj:=wobjEtna;
    TriggL T1693,vl,laserOFF,z0,toolEtna\WObj:=wobjEtna;
    TriggL T1694,v50,laserON,z0,toolEtna\WObj:=wobjEtna;
    TriggL T1695,vl,laserOFF,z0,toolEtna\WObj:=wobjEtna;
    TriggL T1696,v50,laserON,z0,toolEtna\WObj:=wobjEtna;
    TriggL T1697,vl,laserOFF,z0,toolEtna\WObj:=wobjEtna;
    TriggL T1698,v50,laserON,z0,toolEtna\WObj:=wobjEtna;
    TriggL T1699,vl,laserOFF,z0,toolEtna\WObj:=wobjEtna;
    TriggL T1700,v50,laserON,z0,toolEtna\WObj:=wobjEtna;
    TriggL T1701,vl,laserOFF,z0,toolEtna\WObj:=wobjEtna;
    TriggL T1702,v50,laserON,z0,toolEtna\WObj:=wobjEtna;
    TriggL T1703,vl,laserOFF,z0,toolEtna\WObj:=wobjEtna;
    TriggL T1704,v50,laserON,z0,toolEtna\WObj:=wobjEtna;
    TriggL T1705,vl,laserOFF,z0,toolEtna\WObj:=wobjEtna;
    TriggL T1706,v50,laserON,z0,toolEtna\WObj:=wobjEtna;
    TriggL T1707,vl,laserOFF,z0,toolEtna\WObj:=wobjEtna;
    TriggL T1708,v50,laserON,z0,toolEtna\WObj:=wobjEtna;
    TriggL T1709,vl,laserOFF,z0,toolEtna\WObj:=wobjEtna;
    TriggL T1710,v50,laserON,z0,toolEtna\WObj:=wobjEtna;
    TriggL T1711,vl,laserOFF,z0,toolEtna\WObj:=wobjEtna;
    TriggL T1712,v50,laserON,z0,toolEtna\WObj:=wobjEtna;
    TriggL T1713,vl,laserOFF,z0,toolEtna\WObj:=wobjEtna;
    TriggL T1714,v50,laserON,z0,toolEtna\WObj:=wobjEtna;
    TriggL T1715,vl,laserOFF,z0,toolEtna\WObj:=wobjEtna;
    TriggL T1716,v50,laserON,z0,toolEtna\WObj:=wobjEtna;
    TriggL T1717,vl,laserOFF,z0,toolEtna\WObj:=wobjEtna;
    TriggL T1718,v50,laserON,z0,toolEtna\WObj:=wobjEtna;
    TriggL T1719,vl,laserOFF,z0,toolEtna\WObj:=wobjEtna;
    TriggL T1720,v50,laserON,z0,toolEtna\WObj:=wobjEtna;
    TriggL T1721,vl,laserOFF,z0,toolEtna\WObj:=wobjEtna;
    TriggL T1722,v50,laserON,z0,toolEtna\WObj:=wobjEtna;
    TriggL T1723,vl,laserOFF,z0,toolEtna\WObj:=wobjEtna;
    TriggL T1724,v50,laserON,z0,toolEtna\WObj:=wobjEtna;
    TriggL T1725,vl,laserOFF,z0,toolEtna\WObj:=wobjEtna;
    TriggL T1726,v50,laserON,z0,toolEtna\WObj:=wobjEtna;
    TriggL T1727,vl,laserOFF,z0,toolEtna\WObj:=wobjEtna;
    TriggL T1728,v50,laserON,z0,toolEtna\WObj:=wobjEtna;
    TriggL T1729,vl,laserOFF,z0,toolEtna\WObj:=wobjEtna;
    TriggL T1730,v50,laserON,z0,toolEtna\WObj:=wobjEtna;
    TriggL T1731,vl,laserOFF,z0,toolEtna\WObj:=wobjEtna;
    TriggL T1732,v50,laserON,z0,toolEtna\WObj:=wobjEtna;
    TriggL T1733,vl,laserOFF,z0,toolEtna\WObj:=wobjEtna;
    TriggL T1734,v50,laserON,z0,toolEtna\WObj:=wobjEtna;
    TriggL T1735,vl,laserOFF,z0,toolEtna\WObj:=wobjEtna;
    TriggL T1736,v50,laserON,z0,toolEtna\WObj:=wobjEtna;
    TriggL T1737,vl,laserOFF,z0,toolEtna\WObj:=wobjEtna;
    TriggL T1738,v50,laserON,z0,toolEtna\WObj:=wobjEtna;
    TriggL T1739,vl,laserOFF,z0,toolEtna\WObj:=wobjEtna;
    TriggL T1740,v50,laserON,z0,toolEtna\WObj:=wobjEtna;
    TriggL T1741,vl,laserOFF,z0,toolEtna\WObj:=wobjEtna;
    TriggL T1742,v50,laserON,z0,toolEtna\WObj:=wobjEtna;
    TriggL T1743,vl,laserOFF,z0,toolEtna\WObj:=wobjEtna;
    TriggL T1744,v50,laserON,z0,toolEtna\WObj:=wobjEtna;
    TriggL T1745,vl,laserOFF,z0,toolEtna\WObj:=wobjEtna;
    TriggL T1746,v50,laserON,z0,toolEtna\WObj:=wobjEtna;
    TriggL T1747,vl,laserOFF,z0,toolEtna\WObj:=wobjEtna;
    TriggL T1748,v50,laserON,z0,toolEtna\WObj:=wobjEtna;
    TriggL T1749,vl,laserOFF,z0,toolEtna\WObj:=wobjEtna;
    TriggL T1750,v50,laserON,z0,toolEtna\WObj:=wobjEtna;
    TriggL T1751,vl,laserOFF,z0,toolEtna\WObj:=wobjEtna;
    TriggL T1752,v50,laserON,z0,toolEtna\WObj:=wobjEtna;
    TriggL T1753,vl,laserOFF,z0,toolEtna\WObj:=wobjEtna;
    TriggL T1754,v50,laserON,z0,toolEtna\WObj:=wobjEtna;
    TriggL T1755,vl,laserOFF,z0,toolEtna\WObj:=wobjEtna;
    TriggL T1756,v50,laserON,z0,toolEtna\WObj:=wobjEtna;
    TriggL T1757,vl,laserOFF,z0,toolEtna\WObj:=wobjEtna;
    TriggL T1758,v50,laserON,z0,toolEtna\WObj:=wobjEtna;
    TriggL T1759,vl,laserOFF,z0,toolEtna\WObj:=wobjEtna;
    TriggL T1760,v50,laserON,z0,toolEtna\WObj:=wobjEtna;
    TriggL T1761,vl,laserOFF,z0,toolEtna\WObj:=wobjEtna;
    TriggL T1762,v50,laserON,z0,toolEtna\WObj:=wobjEtna;
    TriggL T1763,vl,laserOFF,z0,toolEtna\WObj:=wobjEtna;
    TriggL T1764,v50,laserON,z0,toolEtna\WObj:=wobjEtna;
    TriggL T1765,vl,laserOFF,z0,toolEtna\WObj:=wobjEtna;
    TriggL T1766,v50,laserON,z0,toolEtna\WObj:=wobjEtna;
    TriggL T1767,vl,laserOFF,z0,toolEtna\WObj:=wobjEtna;
    TriggL T1768,v50,laserON,z0,toolEtna\WObj:=wobjEtna;
    TriggL T1769,vl,laserOFF,z0,toolEtna\WObj:=wobjEtna;
    TriggL T1770,v50,laserON,z0,toolEtna\WObj:=wobjEtna;
    TriggL T1771,vl,laserOFF,z0,toolEtna\WObj:=wobjEtna;
    TriggL T1772,v50,laserON,z0,toolEtna\WObj:=wobjEtna;
